LIN {X 0,Y 524.001,Z 252.027,A -85,B 0,C 180,E1 -4869.26,E2 -4869.26} C_VEL
LIN {X 0,Y 524.005,Z 252.027,A -85,B 0,C 180,E1 -4871.738,E2 -4871.738} C_VEL
LIN {X 0,Y 523.995,Z 252.029,A -85,B 0,C 180,E1 -4875.051,E2 -4875.051} C_VEL
LIN {X 0,Y 523.965,Z 252.033,A -85,B 0,C 180,E1 -4877.967,E2 -4877.967} C_VEL
LIN {X 0,Y 523.972,Z 252.031,A -85,B 0,C 180,E1 -4880.408,E2 -4880.408} C_VEL
LIN {X 0,Y 523.916,Z 252.038,A -85,B 0,C 180,E1 -4882.891,E2 -4882.891} C_VEL
LIN {X 0,Y 523.951,Z 252.035,A -85,B 0,C 180,E1 -4885.417,E2 -4885.417} C_VEL
LIN {X 0,Y 523.968,Z 252.033,A -85,B 0,C 180,E1 -4887.997,E2 -4887.997} C_VEL
LIN {X 0,Y 523.943,Z 252.034,A -85,B 0,C 180,E1 -4890.853,E2 -4890.853} C_VEL
LIN {X 0,Y 523.958,Z 252.033,A -85,B 0,C 180,E1 -4893.733,E2 -4893.733} C_VEL
LIN {X 0,Y 523.917,Z 252.038,A -85,B 0,C 180,E1 -4896.402,E2 -4896.402} C_VEL
LIN {X 0,Y 523.925,Z 252.037,A -85,B 0,C 180,E1 -4899.082,E2 -4899.082} C_VEL
LIN {X 0,Y 523.965,Z 252.034,A -85,B 0,C 180,E1 -4901.31,E2 -4901.31} C_VEL
LIN {X 0,Y 523.947,Z 252.035,A -85,B 0,C 180,E1 -4904.689,E2 -4904.689} C_VEL
LIN {X 0,Y 523.916,Z 252.038,A -85,B 0,C 180,E1 -4906.898,E2 -4906.898} C_VEL
LIN {X 0,Y 523.251,Z 252.122,A -85,B 0,C 180,E1 -4907.539,E2 -4907.539} C_VEL
LIN {X 0,Y 520.416,Z 252.476,A -85,B 0,C 180,E1 -4908.581,E2 -4908.581} C_VEL
LIN {X 0,Y 518.018,Z 252.775,A -85,B 0,C 180,E1 -4909.42,E2 -4909.42} C_VEL
LIN {X 0,Y 516.986,Z 252.902,A -85,B 0,C 180,E1 -4910.068,E2 -4910.068} C_VEL
LIN {X 0,Y 516.9,Z 252.911,A -85,B 0,C 180,E1 -4910.287,E2 -4910.287} C_VEL
LIN {X 0,Y 516.875,Z 252.916,A -85,B 0,C 180,E1 -4913.339,E2 -4913.339} C_VEL
LIN {X 0,Y 516.901,Z 252.911,A -85,B 0,C 180,E1 -4916.119,E2 -4916.119} C_VEL
LIN {X 0,Y 516.881,Z 252.915,A -85,B 0,C 180,E1 -4918.933,E2 -4918.933} C_VEL
LIN {X 0,Y 516.911,Z 252.911,A -85,B 0,C 180,E1 -4921.583,E2 -4921.583} C_VEL
LIN {X 0,Y 516.918,Z 252.91,A -85,B 0,C 180,E1 -4924.209,E2 -4924.209} C_VEL
LIN {X 0,Y 516.88,Z 252.916,A -85,B 0,C 180,E1 -4926.776,E2 -4926.776} C_VEL
LIN {X 0,Y 516.923,Z 252.91,A -85,B 0,C 180,E1 -4929.73,E2 -4929.73} C_VEL
LIN {X 0,Y 516.734,Z 252.935,A -85,B 0,C 180,E1 -4932.588,E2 -4932.588} C_VEL
LIN {X 0,Y 516.57,Z 252.955,A -85,B 0,C 180,E1 -4933.398,E2 -4933.398} C_VEL
LIN {X 0,Y 516.586,Z 256.109,A -85,B 0,C 180,E1 -4935.824,E2 -4935.824} C_VEL
LIN {X 0,Y 516.629,Z 259.54,A -85,B 0,C 180,E1 -4938.354,E2 -4938.354} C_VEL
LIN {X 0,Y 516.52,Z 263.691,A -85,B 0,C 180,E1 -4941.391,E2 -4941.391} C_VEL
LIN {X 0,Y 516.557,Z 266.915,A -85,B 0,C 180,E1 -4943.75,E2 -4943.75} C_VEL
LIN {X 0,Y 516.536,Z 270.185,A -85,B 0,C 180,E1 -4946.098,E2 -4946.098} C_VEL
LIN {X 0,Y 516.329,Z 274.545,A -85,B 0,C 180,E1 -4949.219,E2 -4949.219} C_VEL
LIN {X 0,Y 516.246,Z 279.024,A -85,B 0,C 180,E1 -4952.34,E2 -4952.34} C_VEL
LIN {X 0,Y 516.345,Z 280.192,A -85,B 0,C 180,E1 -4953.144,E2 -4953.144} C_VEL
LIN {X 0,Y 517.624,Z 289.128,A -85,B 0,C 180,E1 -4953.453,E2 -4953.453} C_VEL
LIN {X 0,Y 517.444,Z 299.239,A -85,B 0,C 180,E1 -4953.893,E2 -4953.893} C_VEL
LIN {X 0,Y 517.24,Z 307.848,A -85,B 0,C 180,E1 -4954.382,E2 -4954.382} C_VEL
LIN {X 0,Y 517.051,Z 316.077,A -85,B 0,C 180,E1 -4954.97,E2 -4954.97} C_VEL
LIN {X 0,Y 516.884,Z 323.872,A -85,B 0,C 180,E1 -4955.656,E2 -4955.656} C_VEL
LIN {X 0,Y 516.785,Z 331.136,A -85,B 0,C 180,E1 -4956.439,E2 -4956.439} C_VEL
LIN {X 0,Y 516.64,Z 338.552,A -85,B 0,C 180,E1 -4957.424,E2 -4957.424} C_VEL
LIN {X 0,Y 516.488,Z 344.371,A -85,B 0,C 180,E1 -4958.41,E2 -4958.41} C_VEL
LIN {X 0,Y 516.371,Z 348.963,A -85,B 0,C 180,E1 -4959.399,E2 -4959.399} C_VEL
LIN {X 0,Y 516.352,Z 351.937,A -85,B 0,C 180,E1 -4960.191,E2 -4960.191} C_VEL
LIN {X 0,Y 516.316,Z 354.262,A -85,B 0,C 180,E1 -4960.985,E2 -4960.985} C_VEL
LIN {X 0,Y 516.276,Z 355.976,A -85,B 0,C 180,E1 -4961.781,E2 -4961.781} C_VEL
LIN {X 0,Y 516.227,Z 357.177,A -85,B 0,C 180,E1 -4962.58,E2 -4962.58} C_VEL
LIN {X 0,Y 516.198,Z 357.883,A -85,B 0,C 180,E1 -4963.382,E2 -4963.382} C_VEL
LIN {X 0,Y 516.219,Z 358.098,A -85,B 0,C 180,E1 -4964.184,E2 -4964.184} C_VEL
LIN {X 0,Y 516.216,Z 357.765,A -85,B 0,C 180,E1 -4964.99,E2 -4964.99} C_VEL
LIN {X 0,Y 516.236,Z 356.832,A -85,B 0,C 180,E1 -4965.799,E2 -4965.799} C_VEL
LIN {X 0,Y 516.287,Z 354.51,A -85,B 0,C 180,E1 -4967.017,E2 -4967.017} C_VEL
LIN {X 0,Y 516.374,Z 350.713,A -85,B 0,C 180,E1 -4968.241,E2 -4968.241} C_VEL
LIN {X 0,Y 516.445,Z 347.395,A -85,B 0,C 180,E1 -4969.061,E2 -4969.061} C_VEL
LIN {X 0,Y 516.519,Z 343.292,A -85,B 0,C 180,E1 -4969.885,E2 -4969.885} C_VEL
LIN {X 0,Y 516.65,Z 336.774,A -85,B 0,C 180,E1 -4970.92,E2 -4970.92} C_VEL
LIN {X 0,Y 516.798,Z 330.309,A -85,B 0,C 180,E1 -4971.75,E2 -4971.75} C_VEL
LIN {X 0,Y 516.93,Z 324.106,A -85,B 0,C 180,E1 -4972.413,E2 -4972.413} C_VEL
LIN {X 0,Y 517.124,Z 316.421,A -85,B 0,C 180,E1 -4973.094,E2 -4973.094} C_VEL
LIN {X 0,Y 517.321,Z 309.115,A -85,B 0,C 180,E1 -4973.625,E2 -4973.625} C_VEL
LIN {X 0,Y 517.474,Z 300.931,A -85,B 0,C 180,E1 -4974.109,E2 -4974.109} C_VEL
LIN {X 0,Y 517.594,Z 291.635,A -85,B 0,C 180,E1 -4974.537,E2 -4974.537} C_VEL
LIN {X 0,Y 517.263,Z 285.961,A -85,B 0,C 180,E1 -4974.75,E2 -4974.75} C_VEL
LIN {X 0,Y 516.275,Z 280.189,A -85,B 0,C 180,E1 -4974.96,E2 -4974.96} C_VEL
LIN {X 0,Y 516.296,Z 275.269,A -85,B 0,C 180,E1 -4978.451,E2 -4978.451} C_VEL
LIN {X 0,Y 516.338,Z 271.494,A -85,B 0,C 180,E1 -4981.145,E2 -4981.145} C_VEL
LIN {X 0,Y 516.359,Z 267.678,A -85,B 0,C 180,E1 -4983.919,E2 -4983.919} C_VEL
LIN {X 0,Y 516.405,Z 263.771,A -85,B 0,C 180,E1 -4986.784,E2 -4986.784} C_VEL
LIN {X 0,Y 516.448,Z 259.768,A -85,B 0,C 180,E1 -4989.76,E2 -4989.76} C_VEL
LIN {X 0,Y 516.585,Z 255.637,A -85,B 0,C 180,E1 -4992.86,E2 -4992.86} C_VEL
LIN {X 0,Y 516.633,Z 252.947,A -85,B 0,C 180,E1 -4995.02,E2 -4995.02} C_VEL
LIN {X 0,Y 516.837,Z 252.916,A -85,B 0,C 180,E1 -4997.246,E2 -4997.246} C_VEL
LIN {X 0,Y 516.887,Z 252.916,A -85,B 0,C 180,E1 -4999.587,E2 -4999.587} C_VEL
LIN {X 0,Y 516.85,Z 252.917,A -85,B 0,C 180,E1 -5002.276,E2 -5002.276} C_VEL
LIN {X 0,Y 516.876,Z 252.912,A -85,B 0,C 180,E1 -5005.177,E2 -5005.177} C_VEL
LIN {X 0,Y 516.856,Z 252.915,A -85,B 0,C 180,E1 -5007.976,E2 -5007.976} C_VEL
LIN {X 0,Y 516.904,Z 252.912,A -85,B 0,C 180,E1 -5010.697,E2 -5010.697} C_VEL
LIN {X 0,Y 516.925,Z 252.91,A -85,B 0,C 180,E1 -5013.805,E2 -5013.805} C_VEL
LIN {X 0,Y 516.847,Z 252.918,A -85,B 0,C 180,E1 -5016.777,E2 -5016.777} C_VEL
LIN {X 0,Y 516.923,Z 252.906,A -85,B 0,C 180,E1 -5019.733,E2 -5019.733} C_VEL
LIN {X 0,Y 516.915,Z 252.905,A -85,B 0,C 180,E1 -5022.598,E2 -5022.598} C_VEL
LIN {X 0,Y 516.925,Z 252.908,A -85,B 0,C 180,E1 -5025.031,E2 -5025.031} C_VEL
LIN {X 0,Y 516.99,Z 252.9,A -85,B 0,C 180,E1 -5028.236,E2 -5028.236} C_VEL
LIN {X 0,Y 516.953,Z 252.905,A -85,B 0,C 180,E1 -5031.401,E2 -5031.401} C_VEL
LIN {X 0,Y 517.009,Z 252.898,A -85,B 0,C 180,E1 -5034.541,E2 -5034.541} C_VEL
LIN {X 0,Y 517.074,Z 252.89,A -85,B 0,C 180,E1 -5037.665,E2 -5037.665} C_VEL
LIN {X 0,Y 517.082,Z 252.89,A -85,B 0,C 180,E1 -5040.78,E2 -5040.78} C_VEL
LIN {X 0,Y 517.001,Z 252.896,A -85,B 0,C 180,E1 -5043.118,E2 -5043.118} C_VEL
LIN {X 0,Y 517.002,Z 252.894,A -85,B 0,C 180,E1 -5046.245,E2 -5046.245} C_VEL
LIN {X 0,Y 516.933,Z 252.904,A -85,B 0,C 180,E1 -5049.391,E2 -5049.391} C_VEL
LIN {X 0,Y 516.974,Z 252.905,A -85,B 0,C 180,E1 -5051.825,E2 -5051.825} C_VEL
LIN {X 0,Y 516.935,Z 252.908,A -85,B 0,C 180,E1 -5055.148,E2 -5055.148} C_VEL
LIN {X 0,Y 516.903,Z 252.913,A -85,B 0,C 180,E1 -5058.224,E2 -5058.224} C_VEL
LIN {X 0,Y 516.903,Z 252.909,A -85,B 0,C 180,E1 -5060.703,E2 -5060.703} C_VEL
LIN {X 0,Y 516.904,Z 252.91,A -85,B 0,C 180,E1 -5064.073,E2 -5064.073} C_VEL
LIN {X 0,Y 516.889,Z 252.911,A -85,B 0,C 180,E1 -5066.661,E2 -5066.661} C_VEL
LIN {X 0,Y 516.903,Z 252.912,A -85,B 0,C 180,E1 -5069.525,E2 -5069.525} C_VEL
LIN {X 0,Y 516.894,Z 252.915,A -85,B 0,C 180,E1 -5072.546,E2 -5072.546} C_VEL
LIN {X 0,Y 516.857,Z 252.919,A -85,B 0,C 180,E1 -5075.331,E2 -5075.331} C_VEL
LIN {X 0,Y 516.88,Z 252.917,A -85,B 0,C 180,E1 -5078.717,E2 -5078.717} C_VEL
LIN {X 0,Y 516.911,Z 252.912,A -85,B 0,C 180,E1 -5081.776,E2 -5081.776} C_VEL
LIN {X 0,Y 516.89,Z 252.918,A -85,B 0,C 180,E1 -5085.008,E2 -5085.008} C_VEL
LIN {X 0,Y 516.913,Z 252.912,A -85,B 0,C 180,E1 -5088.4,E2 -5088.4} C_VEL
LIN {X 0,Y 516.875,Z 252.917,A -85,B 0,C 180,E1 -5091.285,E2 -5091.285} C_VEL
LIN {X 0,Y 516.869,Z 252.918,A -85,B 0,C 180,E1 -5094.221,E2 -5094.221} C_VEL
LIN {X 0,Y 516.898,Z 252.925,A -85,B 0,C 180,E1 -5094.898,E2 -5094.898} C_VEL
LIN {X 0,Y 517.688,Z 257.17,A -85,B 0,C 180,E1 -5096.647,E2 -5096.647} C_VEL
LIN {X 0,Y 517.651,Z 262.78,A -85,B 0,C 180,E1 -5098.797,E2 -5098.797} C_VEL
LIN {X 0,Y 517.346,Z 271.703,A -85,B 0,C 180,E1 -5102.008,E2 -5102.008} C_VEL
LIN {X 0,Y 517.053,Z 280.514,A -85,B 0,C 180,E1 -5105.081,E2 -5105.081} C_VEL
LIN {X 0,Y 516.846,Z 289.348,A -85,B 0,C 180,E1 -5108.042,E2 -5108.042} C_VEL
LIN {X 0,Y 516.671,Z 299.586,A -85,B 0,C 180,E1 -5111.359,E2 -5111.359} C_VEL
LIN {X 0,Y 516.561,Z 309.871,A -85,B 0,C 180,E1 -5114.616,E2 -5114.616} C_VEL
LIN {X 0,Y 516.453,Z 320.168,A -85,B 0,C 180,E1 -5117.824,E2 -5117.824} C_VEL
LIN {X 0,Y 516.452,Z 324.035,A -85,B 0,C 180,E1 -5119.018,E2 -5119.018} C_VEL
LIN {X 0,Y 517.543,Z 335.925,A -85,B 0,C 180,E1 -5119.388,E2 -5119.388} C_VEL
LIN {X 0,Y 517.369,Z 346.244,A -85,B 0,C 180,E1 -5119.83,E2 -5119.83} C_VEL
LIN {X 0,Y 517.182,Z 354.979,A -85,B 0,C 180,E1 -5120.32,E2 -5120.32} C_VEL
LIN {X 0,Y 516.995,Z 363.323,A -85,B 0,C 180,E1 -5120.909,E2 -5120.909} C_VEL
LIN {X 0,Y 516.826,Z 371.224,A -85,B 0,C 180,E1 -5121.595,E2 -5121.595} C_VEL
LIN {X 0,Y 516.652,Z 378.613,A -85,B 0,C 180,E1 -5122.38,E2 -5122.38} C_VEL
LIN {X 0,Y 516.528,Z 385.999,A -85,B 0,C 180,E1 -5123.343,E2 -5123.343} C_VEL
LIN {X 0,Y 516.449,Z 392.004,A -85,B 0,C 180,E1 -5124.339,E2 -5124.339} C_VEL
LIN {X 0,Y 516.312,Z 396.638,A -85,B 0,C 180,E1 -5125.316,E2 -5125.316} C_VEL
LIN {X 0,Y 516.361,Z 399.657,A -85,B 0,C 180,E1 -5126.099,E2 -5126.099} C_VEL
LIN {X 0,Y 516.294,Z 401.992,A -85,B 0,C 180,E1 -5126.88,E2 -5126.88} C_VEL
LIN {X 0,Y 516.263,Z 403.75,A -85,B 0,C 180,E1 -5127.66,E2 -5127.66} C_VEL
LIN {X 0,Y 516.191,Z 405.007,A -85,B 0,C 180,E1 -5128.441,E2 -5128.441} C_VEL
LIN {X 0,Y 516.16,Z 405.791,A -85,B 0,C 180,E1 -5129.221,E2 -5129.221} C_VEL
LIN {X 0,Y 516.16,Z 406.089,A -85,B 0,C 180,E1 -5130.001,E2 -5130.001} C_VEL
LIN {X 0,Y 516.16,Z 405.792,A -85,B 0,C 180,E1 -5130.781,E2 -5130.781} C_VEL
LIN {X 0,Y 516.191,Z 405.009,A -85,B 0,C 180,E1 -5131.561,E2 -5131.561} C_VEL
LIN {X 0,Y 516.263,Z 403.752,A -85,B 0,C 180,E1 -5132.342,E2 -5132.342} C_VEL
LIN {X 0,Y 516.323,Z 400.836,A -85,B 0,C 180,E1 -5133.513,E2 -5133.513} C_VEL
LIN {X 0,Y 516.342,Z 398.176,A -85,B 0,C 180,E1 -5134.294,E2 -5134.294} C_VEL
LIN {X 0,Y 516.425,Z 392.973,A -85,B 0,C 180,E1 -5135.467,E2 -5135.467} C_VEL
LIN {X 0,Y 516.507,Z 387.575,A -85,B 0,C 180,E1 -5136.414,E2 -5136.414} C_VEL
LIN {X 0,Y 516.626,Z 380.33,A -85,B 0,C 180,E1 -5137.426,E2 -5137.426} C_VEL
LIN {X 0,Y 516.829,Z 372.266,A -85,B 0,C 180,E1 -5138.308,E2 -5138.308} C_VEL
LIN {X 0,Y 516.958,Z 364.569,A -85,B 0,C 180,E1 -5138.996,E2 -5138.996} C_VEL
LIN {X 0,Y 517.141,Z 356.49,A -85,B 0,C 180,E1 -5139.584,E2 -5139.584} C_VEL
LIN {X 0,Y 517.375,Z 348.126,A -85,B 0,C 180,E1 -5140.073,E2 -5140.073} C_VEL
LIN {X 0,Y 517.486,Z 339.588,A -85,B 0,C 180,E1 -5140.467,E2 -5140.467} C_VEL
LIN {X 0,Y 517.348,Z 332.736,A -85,B 0,C 180,E1 -5140.717,E2 -5140.717} C_VEL
LIN {X 0,Y 516.423,Z 324.083,A -85,B 0,C 180,E1 -5140.984,E2 -5140.984} C_VEL
LIN {X 0,Y 516.495,Z 313.787,A -85,B 0,C 180,E1 -5144.178,E2 -5144.178} C_VEL
LIN {X 0,Y 516.569,Z 304.8,A -85,B 0,C 180,E1 -5147.009,E2 -5147.009} C_VEL
LIN {X 0,Y 516.707,Z 295.849,A -85,B 0,C 180,E1 -5149.88,E2 -5149.88} C_VEL
LIN {X 0,Y 516.931,Z 286.915,A -85,B 0,C 180,E1 -5152.798,E2 -5152.798} C_VEL
LIN {X 0,Y 517.115,Z 278.013,A -85,B 0,C 180,E1 -5155.78,E2 -5155.78} C_VEL
LIN {X 0,Y 517.404,Z 269.157,A -85,B 0,C 180,E1 -5158.83,E2 -5158.83} C_VEL
LIN {X 0,Y 517.663,Z 260.359,A -85,B 0,C 180,E1 -5161.971,E2 -5161.971} C_VEL
LIN {X 0,Y 517.557,Z 256.603,A -85,B 0,C 180,E1 -5163.365,E2 -5163.365} C_VEL
LIN {X 0,Y 516.905,Z 252.913,A -85,B 0,C 180,E1 -5164.824,E2 -5164.824} C_VEL
LIN {X 0,Y 516.887,Z 252.914,A -85,B 0,C 180,E1 -5167.943,E2 -5167.943} C_VEL
LIN {X 0,Y 516.89,Z 252.913,A -85,B 0,C 180,E1 -5170.742,E2 -5170.742} C_VEL
LIN {X 0,Y 516.89,Z 252.912,A -85,B 0,C 180,E1 -5172.832,E2 -5172.832} C_VEL
LIN {X 0,Y 516.903,Z 252.91,A -85,B 0,C 180,E1 -5175.007,E2 -5175.007} C_VEL
LIN {X 0,Y 516.921,Z 252.911,A -85,B 0,C 180,E1 -5178.399,E2 -5178.399} C_VEL
LIN {X 0,Y 516.887,Z 252.914,A -85,B 0,C 180,E1 -5181.284,E2 -5181.284} C_VEL
LIN {X 0,Y 516.876,Z 252.916,A -85,B 0,C 180,E1 -5184.219,E2 -5184.219} C_VEL
LIN {X 0,Y 516.903,Z 252.911,A -85,B 0,C 180,E1 -5187.053,E2 -5187.053} C_VEL
LIN {X 0,Y 516.9,Z 252.913,A -85,B 0,C 180,E1 -5189.796,E2 -5189.796} C_VEL
LIN {X 0,Y 516.933,Z 252.908,A -85,B 0,C 180,E1 -5192.467,E2 -5192.467} C_VEL
LIN {X 0,Y 516.884,Z 252.914,A -85,B 0,C 180,E1 -5195.07,E2 -5195.07} C_VEL
LIN {X 0,Y 516.877,Z 252.917,A -85,B 0,C 180,E1 -5197.621,E2 -5197.621} C_VEL
LIN {X 0,Y 516.94,Z 252.906,A -85,B 0,C 180,E1 -5200.129,E2 -5200.129} C_VEL
LIN {X 0,Y 516.913,Z 252.91,A -85,B 0,C 180,E1 -5202.595,E2 -5202.595} C_VEL
LIN {X 0,Y 516.949,Z 252.907,A -85,B 0,C 180,E1 -5205.029,E2 -5205.029} C_VEL
LIN {X 0,Y 516.974,Z 252.902,A -85,B 0,C 180,E1 -5208.233,E2 -5208.233} C_VEL
LIN {X 0,Y 516.962,Z 252.904,A -85,B 0,C 180,E1 -5211.398,E2 -5211.398} C_VEL
LIN {X 0,Y 517.007,Z 252.899,A -85,B 0,C 180,E1 -5213.756,E2 -5213.756} C_VEL
LIN {X 0,Y 517.018,Z 252.899,A -85,B 0,C 180,E1 -5216.882,E2 -5216.882} C_VEL
LIN {X 0,Y 517.09,Z 252.889,A -85,B 0,C 180,E1 -5219.999,E2 -5219.999} C_VEL
LIN {X 0,Y 517.018,Z 252.897,A -85,B 0,C 180,E1 -5223.115,E2 -5223.115} C_VEL
LIN {X 0,Y 517.015,Z 252.899,A -85,B 0,C 180,E1 -5226.242,E2 -5226.242} C_VEL
LIN {X 0,Y 516.955,Z 252.905,A -85,B 0,C 180,E1 -5229.388,E2 -5229.388} C_VEL
LIN {X 0,Y 516.955,Z 252.905,A -85,B 0,C 180,E1 -5231.805,E2 -5231.805} C_VEL
LIN {X 0,Y 516.946,Z 252.907,A -85,B 0,C 180,E1 -5235.145,E2 -5235.145} C_VEL
LIN {X 0,Y 516.926,Z 252.91,A -85,B 0,C 180,E1 -5238.22,E2 -5238.22} C_VEL
LIN {X 0,Y 516.912,Z 252.91,A -85,B 0,C 180,E1 -5240.7,E2 -5240.7} C_VEL
LIN {X 0,Y 516.91,Z 252.912,A -85,B 0,C 180,E1 -5244.07,E2 -5244.07} C_VEL
LIN {X 0,Y 516.925,Z 252.908,A -85,B 0,C 180,E1 -5246.656,E2 -5246.656} C_VEL
LIN {X 0,Y 516.908,Z 252.912,A -85,B 0,C 180,E1 -5249.522,E2 -5249.522} C_VEL
LIN {X 0,Y 516.897,Z 252.912,A -85,B 0,C 180,E1 -5252.542,E2 -5252.542} C_VEL
LIN {X 0,Y 516.878,Z 252.917,A -85,B 0,C 180,E1 -5255.33,E2 -5255.33} C_VEL
LIN {X 0,Y 516.875,Z 252.915,A -85,B 0,C 180,E1 -5257.941,E2 -5257.941} C_VEL
LIN {X 0,Y 516.897,Z 252.913,A -85,B 0,C 180,E1 -5260.738,E2 -5260.738} C_VEL
LIN {X 0,Y 516.874,Z 252.915,A -85,B 0,C 180,E1 -5263.901,E2 -5263.901} C_VEL
LIN {X 0,Y 516.874,Z 252.915,A -85,B 0,C 180,E1 -5266.105,E2 -5266.105} C_VEL
LIN {X 0,Y 516.898,Z 252.913,A -85,B 0,C 180,E1 -5269.259,E2 -5269.259} C_VEL
LIN {X 0,Y 516.9,Z 252.911,A -85,B 0,C 180,E1 -5270.287,E2 -5270.287} C_VEL
LIN {X 0,Y 516.23,Z 252.996,A -85,B 0,C 180,E1 -5270.937,E2 -5270.937} C_VEL
LIN {X 0,Y 513.374,Z 253.353,A -85,B 0,C 180,E1 -5271.992,E2 -5271.992} C_VEL
LIN {X 0,Y 510.957,Z 253.655,A -85,B 0,C 180,E1 -5272.842,E2 -5272.842} C_VEL
LIN {X 0,Y 509.911,Z 253.784,A -85,B 0,C 180,E1 -5273.498,E2 -5273.498} C_VEL
LIN {X 0,Y 509.822,Z 253.793,A -85,B 0,C 180,E1 -5273.721,E2 -5273.721} C_VEL
LIN {X 0,Y 509.851,Z 253.791,A -85,B 0,C 180,E1 -5276.538,E2 -5276.538} C_VEL
LIN {X 0,Y 509.837,Z 253.793,A -85,B 0,C 180,E1 -5279.333,E2 -5279.333} C_VEL
LIN {X 0,Y 509.881,Z 253.786,A -85,B 0,C 180,E1 -5282.053,E2 -5282.053} C_VEL
LIN {X 0,Y 509.865,Z 253.79,A -85,B 0,C 180,E1 -5284.702,E2 -5284.702} C_VEL
LIN {X 0,Y 509.867,Z 253.788,A -85,B 0,C 180,E1 -5287.441,E2 -5287.441} C_VEL
LIN {X 0,Y 509.899,Z 253.785,A -85,B 0,C 180,E1 -5289.843,E2 -5289.843} C_VEL
LIN {X 0,Y 509.731,Z 253.807,A -85,B 0,C 180,E1 -5292.341,E2 -5292.341} C_VEL
LIN {X 0,Y 509.561,Z 253.827,A -85,B 0,C 180,E1 -5293.163,E2 -5293.163} C_VEL
LIN {X 0,Y 509.492,Z 254.335,A -85,B 0,C 180,E1 -5293.984,E2 -5293.984} C_VEL
LIN {X 0,Y 509.493,Z 257.625,A -85,B 0,C 180,E1 -5296.437,E2 -5296.437} C_VEL
LIN {X 0,Y 509.501,Z 260.888,A -85,B 0,C 180,E1 -5298.864,E2 -5298.864} C_VEL
LIN {X 0,Y 509.425,Z 265.235,A -85,B 0,C 180,E1 -5302.069,E2 -5302.069} C_VEL
LIN {X 0,Y 509.508,Z 267.408,A -85,B 0,C 180,E1 -5303.664,E2 -5303.664} C_VEL
LIN {X 0,Y 509.453,Z 270.692,A -85,B 0,C 180,E1 -5306.044,E2 -5306.044} C_VEL
LIN {X 0,Y 509.252,Z 275.102,A -85,B 0,C 180,E1 -5309.208,E2 -5309.208} C_VEL
LIN {X 0,Y 509.258,Z 280.437,A -85,B 0,C 180,E1 -5312.965,E2 -5312.965} C_VEL
LIN {X 0,Y 510.305,Z 286.696,A -85,B 0,C 180,E1 -5313.206,E2 -5313.206} C_VEL
LIN {X 0,Y 510.627,Z 291.745,A -85,B 0,C 180,E1 -5313.402,E2 -5313.402} C_VEL
LIN {X 0,Y 510.464,Z 299.482,A -85,B 0,C 180,E1 -5313.749,E2 -5313.749} C_VEL
LIN {X 0,Y 510.261,Z 308.102,A -85,B 0,C 180,E1 -5314.245,E2 -5314.245} C_VEL
LIN {X 0,Y 510.059,Z 316.344,A -85,B 0,C 180,E1 -5314.84,E2 -5314.84} C_VEL
LIN {X 0,Y 509.868,Z 324.153,A -85,B 0,C 180,E1 -5315.536,E2 -5315.536} C_VEL
LIN {X 0,Y 509.746,Z 331.438,A -85,B 0,C 180,E1 -5316.331,E2 -5316.331} C_VEL
LIN {X 0,Y 509.606,Z 338.846,A -85,B 0,C 180,E1 -5317.328,E2 -5317.328} C_VEL
LIN {X 0,Y 509.443,Z 344.674,A -85,B 0,C 180,E1 -5318.328,E2 -5318.328} C_VEL
LIN {X 0,Y 509.337,Z 348.485,A -85,B 0,C 180,E1 -5319.129,E2 -5319.129} C_VEL
LIN {X 0,Y 509.272,Z 352.834,A -85,B 0,C 180,E1 -5320.334,E2 -5320.334} C_VEL
LIN {X 0,Y 509.233,Z 355.846,A -85,B 0,C 180,E1 -5321.526,E2 -5321.526} C_VEL
LIN {X 0,Y 509.192,Z 356.701,A -85,B 0,C 180,E1 -5321.947,E2 -5321.947} C_VEL
LIN {X 0,Y 509.136,Z 357.747,A -85,B 0,C 180,E1 -5322.758,E2 -5322.758} C_VEL
LIN {X 0,Y 509.104,Z 358.292,A -85,B 0,C 180,E1 -5323.572,E2 -5323.572} C_VEL
LIN {X 0,Y 509.147,Z 358.126,A -85,B 0,C 180,E1 -5324.94,E2 -5324.94} C_VEL
LIN {X 0,Y 509.164,Z 356.91,A -85,B 0,C 180,E1 -5326.024,E2 -5326.024} C_VEL
LIN {X 0,Y 509.238,Z 354.286,A -85,B 0,C 180,E1 -5327.26,E2 -5327.26} C_VEL
LIN {X 0,Y 509.294,Z 351.801,A -85,B 0,C 180,E1 -5328.099,E2 -5328.099} C_VEL
LIN {X 0,Y 509.366,Z 348.684,A -85,B 0,C 180,E1 -5328.918,E2 -5328.918} C_VEL
LIN {X 0,Y 509.458,Z 343.647,A -85,B 0,C 180,E1 -5329.963,E2 -5329.963} C_VEL
LIN {X 0,Y 509.626,Z 337.138,A -85,B 0,C 180,E1 -5331.01,E2 -5331.01} C_VEL
LIN {X 0,Y 509.77,Z 330.676,A -85,B 0,C 180,E1 -5331.852,E2 -5331.852} C_VEL
LIN {X 0,Y 509.923,Z 323.971,A -85,B 0,C 180,E1 -5332.575,E2 -5332.575} C_VEL
LIN {X 0,Y 510.117,Z 316.671,A -85,B 0,C 180,E1 -5333.226,E2 -5333.226} C_VEL
LIN {X 0,Y 510.324,Z 309.507,A -85,B 0,C 180,E1 -5333.753,E2 -5333.753} C_VEL
LIN {X 0,Y 510.511,Z 300.587,A -85,B 0,C 180,E1 -5334.284,E2 -5334.284} C_VEL
LIN {X 0,Y 510.662,Z 290.756,A -85,B 0,C 180,E1 -5334.731,E2 -5334.731} C_VEL
LIN {X 0,Y 509.759,Z 283.857,A -85,B 0,C 180,E1 -5334.984,E2 -5334.984} C_VEL
LIN {X 0,Y 509.205,Z 280.518,A -85,B 0,C 180,E1 -5335.117,E2 -5335.117} C_VEL
LIN {X 0,Y 509.215,Z 276.475,A -85,B 0,C 180,E1 -5337.985,E2 -5337.985} C_VEL
LIN {X 0,Y 509.262,Z 272.044,A -85,B 0,C 180,E1 -5341.176,E2 -5341.176} C_VEL
LIN {X 0,Y 509.296,Z 268.029,A -85,B 0,C 180,E1 -5344.114,E2 -5344.114} C_VEL
LIN {X 0,Y 509.363,Z 264.365,A -85,B 0,C 180,E1 -5346.849,E2 -5346.849} C_VEL
LIN {X 0,Y 509.382,Z 260.939,A -85,B 0,C 180,E1 -5349.412,E2 -5349.412} C_VEL
LIN {X 0,Y 509.501,Z 256.841,A -85,B 0,C 180,E1 -5352.522,E2 -5352.522} C_VEL
LIN {X 0,Y 509.568,Z 254.029,A -85,B 0,C 180,E1 -5354.698,E2 -5354.698} C_VEL
LIN {X 0,Y 509.794,Z 253.794,A -85,B 0,C 180,E1 -5357.509,E2 -5357.509} C_VEL
LIN {X 0,Y 509.845,Z 253.788,A -85,B 0,C 180,E1 -5360.526,E2 -5360.526} C_VEL
LIN {X 0,Y 509.817,Z 253.792,A -85,B 0,C 180,E1 -5363.649,E2 -5363.649} C_VEL
LIN {X 0,Y 509.842,Z 253.788,A -85,B 0,C 180,E1 -5366.54,E2 -5366.54} C_VEL
LIN {X 0,Y 509.826,Z 253.792,A -85,B 0,C 180,E1 -5369.335,E2 -5369.335} C_VEL
LIN {X 0,Y 509.876,Z 253.787,A -85,B 0,C 180,E1 -5372.056,E2 -5372.056} C_VEL
LIN {X 0,Y 509.858,Z 253.786,A -85,B 0,C 180,E1 -5374.705,E2 -5374.705} C_VEL
LIN {X 0,Y 509.809,Z 253.793,A -85,B 0,C 180,E1 -5377.459,E2 -5377.459} C_VEL
LIN {X 0,Y 509.901,Z 253.782,A -85,B 0,C 180,E1 -5379.846,E2 -5379.846} C_VEL
LIN {X 0,Y 509.87,Z 253.787,A -85,B 0,C 180,E1 -5383.176,E2 -5383.176} C_VEL
LIN {X 0,Y 509.846,Z 253.786,A -85,B 0,C 180,E1 -5385.635,E2 -5385.635} C_VEL
LIN {X 0,Y 509.912,Z 253.778,A -85,B 0,C 180,E1 -5388.876,E2 -5388.876} C_VEL
LIN {X 0,Y 509.936,Z 253.776,A -85,B 0,C 180,E1 -5392.08,E2 -5392.08} C_VEL
LIN {X 0,Y 509.96,Z 253.778,A -85,B 0,C 180,E1 -5394.466,E2 -5394.466} C_VEL
LIN {X 0,Y 510.045,Z 253.765,A -85,B 0,C 180,E1 -5397.632,E2 -5397.632} C_VEL
LIN {X 0,Y 510.052,Z 253.765,A -85,B 0,C 180,E1 -5400.791,E2 -5400.791} C_VEL
LIN {X 0,Y 509.943,Z 253.775,A -85,B 0,C 180,E1 -5403.162,E2 -5403.162} C_VEL
LIN {X 0,Y 509.97,Z 253.77,A -85,B 0,C 180,E1 -5406.331,E2 -5406.331} C_VEL
LIN {X 0,Y 509.901,Z 253.785,A -85,B 0,C 180,E1 -5408.722,E2 -5408.722} C_VEL
LIN {X 0,Y 509.942,Z 253.78,A -85,B 0,C 180,E1 -5411.932,E2 -5411.932} C_VEL
LIN {X 0,Y 509.885,Z 253.785,A -85,B 0,C 180,E1 -5415.243,E2 -5415.243} C_VEL
LIN {X 0,Y 509.852,Z 253.791,A -85,B 0,C 180,E1 -5417.993,E2 -5417.993} C_VEL
LIN {X 0,Y 509.878,Z 253.783,A -85,B 0,C 180,E1 -5420.403,E2 -5420.403} C_VEL
LIN {X 0,Y 509.829,Z 253.79,A -85,B 0,C 180,E1 -5423.565,E2 -5423.565} C_VEL
LIN {X 0,Y 509.876,Z 253.787,A -85,B 0,C 180,E1 -5426.374,E2 -5426.374} C_VEL
LIN {X 0,Y 509.85,Z 253.789,A -85,B 0,C 180,E1 -5429.752,E2 -5429.752} C_VEL
LIN {X 0,Y 509.87,Z 253.788,A -85,B 0,C 180,E1 -5432.776,E2 -5432.776} C_VEL
LIN {X 0,Y 509.816,Z 253.798,A -85,B 0,C 180,E1 -5435.579,E2 -5435.579} C_VEL
LIN {X 0,Y 509.846,Z 253.79,A -85,B 0,C 180,E1 -5438.339,E2 -5438.339} C_VEL
LIN {X 0,Y 509.858,Z 253.787,A -85,B 0,C 180,E1 -5441.426,E2 -5441.426} C_VEL
LIN {X 0,Y 509.834,Z 253.793,A -85,B 0,C 180,E1 -5444.671,E2 -5444.671} C_VEL
LIN {X 0,Y 509.855,Z 253.793,A -85,B 0,C 180,E1 -5448.104,E2 -5448.104} C_VEL
LIN {X 0,Y 509.842,Z 253.79,A -85,B 0,C 180,E1 -5450.649,E2 -5450.649} C_VEL
LIN {X 0,Y 509.821,Z 253.794,A -85,B 0,C 180,E1 -5453.648,E2 -5453.648} C_VEL
LIN {X 0,Y 509.871,Z 253.98,A -85,B 0,C 180,E1 -5454.748,E2 -5454.748} C_VEL
LIN {X 0,Y 510.712,Z 258.417,A -85,B 0,C 180,E1 -5456.604,E2 -5456.604} C_VEL
LIN {X 0,Y 510.706,Z 263.38,A -85,B 0,C 180,E1 -5458.563,E2 -5458.563} C_VEL
LIN {X 0,Y 510.338,Z 272.215,A -85,B 0,C 180,E1 -5461.808,E2 -5461.808} C_VEL
LIN {X 0,Y 510.012,Z 281.573,A -85,B 0,C 180,E1 -5465.123,E2 -5465.123} C_VEL
LIN {X 0,Y 509.774,Z 290.457,A -85,B 0,C 180,E1 -5468.148,E2 -5468.148} C_VEL
LIN {X 0,Y 509.607,Z 299.341,A -85,B 0,C 180,E1 -5471.091,E2 -5471.091} C_VEL
LIN {X 0,Y 509.493,Z 309.604,A -85,B 0,C 180,E1 -5474.397,E2 -5474.397} C_VEL
LIN {X 0,Y 509.342,Z 318.558,A -85,B 0,C 180,E1 -5477.247,E2 -5477.247} C_VEL
LIN {X 0,Y 509.366,Z 323.694,A -85,B 0,C 180,E1 -5478.864,E2 -5478.864} C_VEL
LIN {X 0,Y 510.524,Z 336.827,A -85,B 0,C 180,E1 -5479.291,E2 -5479.291} C_VEL
LIN {X 0,Y 510.361,Z 345.901,A -85,B 0,C 180,E1 -5479.689,E2 -5479.689} C_VEL
LIN {X 0,Y 510.187,Z 354.638,A -85,B 0,C 180,E1 -5480.186,E2 -5480.186} C_VEL
LIN {X 0,Y 509.97,Z 362.983,A -85,B 0,C 180,E1 -5480.782,E2 -5480.782} C_VEL
LIN {X 0,Y 509.799,Z 370.885,A -85,B 0,C 180,E1 -5481.479,E2 -5481.479} C_VEL
LIN {X 0,Y 509.586,Z 378.274,A -85,B 0,C 180,E1 -5482.273,E2 -5482.273} C_VEL
LIN {X 0,Y 509.427,Z 386.444,A -85,B 0,C 180,E1 -5483.368,E2 -5483.368} C_VEL
LIN {X 0,Y 509.342,Z 392.633,A -85,B 0,C 180,E1 -5484.458,E2 -5484.458} C_VEL
LIN {X 0,Y 509.236,Z 397.836,A -85,B 0,C 180,E1 -5485.648,E2 -5485.648} C_VEL
LIN {X 0,Y 509.243,Z 400.499,A -85,B 0,C 180,E1 -5486.44,E2 -5486.44} C_VEL
LIN {X 0,Y 509.192,Z 403.42,A -85,B 0,C 180,E1 -5487.628,E2 -5487.628} C_VEL
LIN {X 0,Y 509.112,Z 404.677,A -85,B 0,C 180,E1 -5488.419,E2 -5488.419} C_VEL
LIN {X 0,Y 509.073,Z 405.461,A -85,B 0,C 180,E1 -5489.21,E2 -5489.21} C_VEL
LIN {X 0,Y 509.071,Z 405.759,A -85,B 0,C 180,E1 -5490.001,E2 -5490.001} C_VEL
LIN {X 0,Y 509.073,Z 405.464,A -85,B 0,C 180,E1 -5490.792,E2 -5490.792} C_VEL
LIN {X 0,Y 509.112,Z 404.681,A -85,B 0,C 180,E1 -5491.583,E2 -5491.583} C_VEL
LIN {X 0,Y 509.192,Z 403.424,A -85,B 0,C 180,E1 -5492.374,E2 -5492.374} C_VEL
LIN {X 0,Y 509.244,Z 400.508,A -85,B 0,C 180,E1 -5493.562,E2 -5493.562} C_VEL
LIN {X 0,Y 509.236,Z 397.846,A -85,B 0,C 180,E1 -5494.354,E2 -5494.354} C_VEL
LIN {X 0,Y 509.342,Z 392.644,A -85,B 0,C 180,E1 -5495.544,E2 -5495.544} C_VEL
LIN {X 0,Y 509.482,Z 386.125,A -85,B 0,C 180,E1 -5496.685,E2 -5496.685} C_VEL
LIN {X 0,Y 509.592,Z 378.294,A -85,B 0,C 180,E1 -5497.729,E2 -5497.729} C_VEL
LIN {X 0,Y 509.801,Z 370.91,A -85,B 0,C 180,E1 -5498.523,E2 -5498.523} C_VEL
LIN {X 0,Y 509.973,Z 363.004,A -85,B 0,C 180,E1 -5499.22,E2 -5499.22} C_VEL
LIN {X 0,Y 510.152,Z 354.654,A -85,B 0,C 180,E1 -5499.817,E2 -5499.817} C_VEL
LIN {X 0,Y 510.424,Z 344,A -85,B 0,C 180,E1 -5500.412,E2 -5500.412} C_VEL
LIN {X 0,Y 510.412,Z 334.072,A -85,B 0,C 180,E1 -5500.814,E2 -5500.814} C_VEL
LIN {X 0,Y 509.327,Z 323.753,A -85,B 0,C 180,E1 -5501.139,E2 -5501.139} C_VEL
LIN {X 0,Y 509.424,Z 314.809,A -85,B 0,C 180,E1 -5503.972,E2 -5503.972} C_VEL
LIN {X 0,Y 509.482,Z 305.849,A -85,B 0,C 180,E1 -5506.84,E2 -5506.84} C_VEL
LIN {X 0,Y 509.629,Z 296.914,A -85,B 0,C 180,E1 -5509.748,E2 -5509.748} C_VEL
LIN {X 0,Y 509.869,Z 287.991,A -85,B 0,C 180,E1 -5512.704,E2 -5512.704} C_VEL
LIN {X 0,Y 510.074,Z 279.105,A -85,B 0,C 180,E1 -5515.724,E2 -5515.724} C_VEL
LIN {X 0,Y 510.288,Z 272.045,A -85,B 0,C 180,E1 -5518.182,E2 -5518.182} C_VEL
LIN {X 0,Y 510.591,Z 264.124,A -85,B 0,C 180,E1 -5521.018,E2 -5521.018} C_VEL
LIN {X 0,Y 510.655,Z 259.011,A -85,B 0,C 180,E1 -5522.909,E2 -5522.909} C_VEL
LIN {X 0,Y 509.864,Z 253.79,A -85,B 0,C 180,E1 -5525.014,E2 -5525.014} C_VEL
LIN {X 0,Y 509.857,Z 253.792,A -85,B 0,C 180,E1 -5528.338,E2 -5528.338} C_VEL
LIN {X 0,Y 509.863,Z 253.789,A -85,B 0,C 180,E1 -5531.426,E2 -5531.426} C_VEL
LIN {X 0,Y 509.847,Z 253.79,A -85,B 0,C 180,E1 -5534.67,E2 -5534.67} C_VEL
LIN {X 0,Y 509.841,Z 253.793,A -85,B 0,C 180,E1 -5537.51,E2 -5537.51} C_VEL
LIN {X 0,Y 509.853,Z 253.79,A -85,B 0,C 180,E1 -5540.647,E2 -5540.647} C_VEL
LIN {X 0,Y 509.817,Z 253.796,A -85,B 0,C 180,E1 -5543.645,E2 -5543.645} C_VEL
LIN {X 0,Y 509.867,Z 253.788,A -85,B 0,C 180,E1 -5546.539,E2 -5546.539} C_VEL
LIN {X 0,Y 509.854,Z 253.79,A -85,B 0,C 180,E1 -5549.334,E2 -5549.334} C_VEL
LIN {X 0,Y 509.898,Z 253.784,A -85,B 0,C 180,E1 -5552.054,E2 -5552.054} C_VEL
LIN {X 0,Y 509.849,Z 253.791,A -85,B 0,C 180,E1 -5554.701,E2 -5554.701} C_VEL
LIN {X 0,Y 509.835,Z 253.793,A -85,B 0,C 180,E1 -5557.457,E2 -5557.457} C_VEL
LIN {X 0,Y 509.925,Z 253.78,A -85,B 0,C 180,E1 -5559.844,E2 -5559.844} C_VEL
LIN {X 0,Y 509.88,Z 253.787,A -85,B 0,C 180,E1 -5563.173,E2 -5563.173} C_VEL
LIN {X 0,Y 509.869,Z 253.789,A -85,B 0,C 180,E1 -5565.633,E2 -5565.633} C_VEL
LIN {X 0,Y 509.919,Z 253.784,A -85,B 0,C 180,E1 -5568.873,E2 -5568.873} C_VEL
LIN {X 0,Y 509.928,Z 253.781,A -85,B 0,C 180,E1 -5572.077,E2 -5572.077} C_VEL
LIN {X 0,Y 509.983,Z 253.774,A -85,B 0,C 180,E1 -5574.463,E2 -5574.463} C_VEL
LIN {X 0,Y 510.06,Z 253.764,A -85,B 0,C 180,E1 -5577.63,E2 -5577.63} C_VEL
LIN {X 0,Y 510.069,Z 253.764,A -85,B 0,C 180,E1 -5580.788,E2 -5580.788} C_VEL
LIN {X 0,Y 509.96,Z 253.776,A -85,B 0,C 180,E1 -5583.159,E2 -5583.159} C_VEL
LIN {X 0,Y 509.983,Z 253.774,A -85,B 0,C 180,E1 -5586.328,E2 -5586.328} C_VEL
LIN {X 0,Y 509.918,Z 253.782,A -85,B 0,C 180,E1 -5588.719,E2 -5588.719} C_VEL
LIN {X 0,Y 509.907,Z 253.784,A -85,B 0,C 180,E1 -5591.93,E2 -5591.93} C_VEL
LIN {X 0,Y 509.896,Z 253.785,A -85,B 0,C 180,E1 -5595.24,E2 -5595.24} C_VEL
LIN {X 0,Y 509.89,Z 253.787,A -85,B 0,C 180,E1 -5597.999,E2 -5597.999} C_VEL
LIN {X 0,Y 509.85,Z 253.79,A -85,B 0,C 180,E1 -5601,E2 -5601} C_VEL
LIN {X 0,Y 509.869,Z 253.788,A -85,B 0,C 180,E1 -5604.424,E2 -5604.424} C_VEL
LIN {X 0,Y 509.884,Z 253.785,A -85,B 0,C 180,E1 -5607.054,E2 -5607.054} C_VEL
LIN {X 0,Y 509.854,Z 253.79,A -85,B 0,C 180,E1 -5609.749,E2 -5609.749} C_VEL
LIN {X 0,Y 509.873,Z 253.786,A -85,B 0,C 180,E1 -5612.773,E2 -5612.773} C_VEL
LIN {X 0,Y 509.838,Z 253.793,A -85,B 0,C 180,E1 -5615.579,E2 -5615.579} C_VEL
LIN {X 0,Y 509.845,Z 253.791,A -85,B 0,C 180,E1 -5618.336,E2 -5618.336} C_VEL
LIN {X 0,Y 509.858,Z 253.791,A -85,B 0,C 180,E1 -5621.422,E2 -5621.422} C_VEL
LIN {X 0,Y 509.848,Z 253.791,A -85,B 0,C 180,E1 -5624.666,E2 -5624.666} C_VEL
LIN {X 0,Y 509.877,Z 253.786,A -85,B 0,C 180,E1 -5628.097,E2 -5628.097} C_VEL
LIN {X 0,Y 509.866,Z 253.79,A -85,B 0,C 180,E1 -5630.648,E2 -5630.648} C_VEL
LIN {X 0,Y 509.822,Z 253.793,A -85,B 0,C 180,E1 -5633.721,E2 -5633.721} C_VEL
LIN {X 0,Y 509.155,Z 253.877,A -85,B 0,C 180,E1 -5634.38,E2 -5634.38} C_VEL
LIN {X 0,Y 506.337,Z 254.229,A -85,B 0,C 180,E1 -5635.452,E2 -5635.452} C_VEL
LIN {X 0,Y 503.944,Z 254.528,A -85,B 0,C 180,E1 -5636.316,E2 -5636.316} C_VEL
LIN {X 0,Y 502.895,Z 254.657,A -85,B 0,C 180,E1 -5636.982,E2 -5636.982} C_VEL
LIN {X 0,Y 502.798,Z 254.667,A -85,B 0,C 180,E1 -5637.208,E2 -5637.208} C_VEL
LIN {X 0,Y 502.817,Z 254.666,A -85,B 0,C 180,E1 -5640.06,E2 -5640.06} C_VEL
LIN {X 0,Y 502.821,Z 254.667,A -85,B 0,C 180,E1 -5642.532,E2 -5642.532} C_VEL
LIN {X 0,Y 502.816,Z 254.666,A -85,B 0,C 180,E1 -5645.296,E2 -5645.296} C_VEL
LIN {X 0,Y 502.804,Z 254.668,A -85,B 0,C 180,E1 -5647.827,E2 -5647.827} C_VEL
LIN {X 0,Y 502.796,Z 254.669,A -85,B 0,C 180,E1 -5650.398,E2 -5650.398} C_VEL
LIN {X 0,Y 502.554,Z 254.7,A -85,B 0,C 180,E1 -5652.921,E2 -5652.921} C_VEL
LIN {X 0,Y 502.437,Z 254.722,A -85,B 0,C 180,E1 -5653.753,E2 -5653.753} C_VEL
LIN {X 0,Y 502.427,Z 258.031,A -85,B 0,C 180,E1 -5656.242,E2 -5656.242} C_VEL
LIN {X 0,Y 502.45,Z 261.322,A -85,B 0,C 180,E1 -5658.706,E2 -5658.706} C_VEL
LIN {X 0,Y 502.371,Z 265.693,A -85,B 0,C 180,E1 -5661.957,E2 -5661.957} C_VEL
LIN {X 0,Y 502.436,Z 267.905,A -85,B 0,C 180,E1 -5663.574,E2 -5663.574} C_VEL
LIN {X 0,Y 502.29,Z 272.316,A -85,B 0,C 180,E1 -5666.791,E2 -5666.791} C_VEL
LIN {X 0,Y 502.108,Z 276.766,A -85,B 0,C 180,E1 -5669.999,E2 -5669.999} C_VEL
LIN {X 0,Y 502.158,Z 280.754,A -85,B 0,C 180,E1 -5672.832,E2 -5672.832} C_VEL
LIN {X 0,Y 503.678,Z 290.767,A -85,B 0,C 180,E1 -5673.198,E2 -5673.198} C_VEL
LIN {X 0,Y 503.487,Z 299.726,A -85,B 0,C 180,E1 -5673.6,E2 -5673.6} C_VEL
LIN {X 0,Y 503.302,Z 308.348,A -85,B 0,C 180,E1 -5674.103,E2 -5674.103} C_VEL
LIN {X 0,Y 503.063,Z 316.613,A -85,B 0,C 180,E1 -5674.707,E2 -5674.707} C_VEL
LIN {X 0,Y 502.87,Z 324.427,A -85,B 0,C 180,E1 -5675.412,E2 -5675.412} C_VEL
LIN {X 0,Y 502.711,Z 331.728,A -85,B 0,C 180,E1 -5676.219,E2 -5676.219} C_VEL
LIN {X 0,Y 502.58,Z 339.138,A -85,B 0,C 180,E1 -5677.229,E2 -5677.229} C_VEL
LIN {X 0,Y 502.406,Z 344.975,A -85,B 0,C 180,E1 -5678.243,E2 -5678.243} C_VEL
LIN {X 0,Y 502.256,Z 349.58,A -85,B 0,C 180,E1 -5679.259,E2 -5679.259} C_VEL
LIN {X 0,Y 502.203,Z 352.565,A -85,B 0,C 180,E1 -5680.073,E2 -5680.073} C_VEL
LIN {X 0,Y 502.164,Z 355.789,A -85,B 0,C 180,E1 -5681.298,E2 -5681.298} C_VEL
LIN {X 0,Y 502.083,Z 357.333,A -85,B 0,C 180,E1 -5682.119,E2 -5682.119} C_VEL
LIN {X 0,Y 502.049,Z 358.311,A -85,B 0,C 180,E1 -5682.942,E2 -5682.942} C_VEL
LIN {X 0,Y 502.025,Z 358.703,A -85,B 0,C 180,E1 -5683.767,E2 -5683.767} C_VEL
LIN {X 0,Y 502.072,Z 358.418,A -85,B 0,C 180,E1 -5685.024,E2 -5685.024} C_VEL
LIN {X 0,Y 502.085,Z 356.881,A -85,B 0,C 180,E1 -5686.256,E2 -5686.256} C_VEL
LIN {X 0,Y 502.167,Z 354.063,A -85,B 0,C 180,E1 -5687.5,E2 -5687.5} C_VEL
LIN {X 0,Y 502.292,Z 349.831,A -85,B 0,C 180,E1 -5688.771,E2 -5688.771} C_VEL
LIN {X 0,Y 502.409,Z 344.105,A -85,B 0,C 180,E1 -5690.023,E2 -5690.023} C_VEL
LIN {X 0,Y 502.576,Z 337.497,A -85,B 0,C 180,E1 -5691.104,E2 -5691.104} C_VEL
LIN {X 0,Y 502.761,Z 331.047,A -85,B 0,C 180,E1 -5691.957,E2 -5691.957} C_VEL
LIN {X 0,Y 502.915,Z 323.852,A -85,B 0,C 180,E1 -5692.739,E2 -5692.739} C_VEL
LIN {X 0,Y 503.153,Z 315.753,A -85,B 0,C 180,E1 -5693.457,E2 -5693.457} C_VEL
LIN {X 0,Y 503.443,Z 304.97,A -85,B 0,C 180,E1 -5694.208,E2 -5694.208} C_VEL
LIN {X 0,Y 503.658,Z 295.451,A -85,B 0,C 180,E1 -5694.697,E2 -5694.697} C_VEL
LIN {X 0,Y 503.478,Z 288.478,A -85,B 0,C 180,E1 -5694.989,E2 -5694.989} C_VEL
LIN {X 0,Y 502.13,Z 280.818,A -85,B 0,C 180,E1 -5695.272,E2 -5695.272} C_VEL
LIN {X 0,Y 502.141,Z 276.453,A -85,B 0,C 180,E1 -5698.414,E2 -5698.414} C_VEL
LIN {X 0,Y 502.184,Z 272.356,A -85,B 0,C 180,E1 -5701.39,E2 -5701.39} C_VEL
LIN {X 0,Y 502.21,Z 268.374,A -85,B 0,C 180,E1 -5704.349,E2 -5704.349} C_VEL
LIN {X 0,Y 502.283,Z 264.686,A -85,B 0,C 180,E1 -5707.107,E2 -5707.107} C_VEL
LIN {X 0,Y 502.326,Z 260.809,A -85,B 0,C 180,E1 -5710.058,E2 -5710.058} C_VEL
LIN {X 0,Y 502.47,Z 256.565,A -85,B 0,C 180,E1 -5713.341,E2 -5713.341} C_VEL
LIN {X 0,Y 502.504,Z 255.069,A -85,B 0,C 180,E1 -5714.501,E2 -5714.501} C_VEL
LIN {X 0,Y 502.576,Z 254.697,A -85,B 0,C 180,E1 -5715.641,E2 -5715.641} C_VEL
LIN {X 0,Y 502.772,Z 254.673,A -85,B 0,C 180,E1 -5717.861,E2 -5717.861} C_VEL
LIN {X 0,Y 502.801,Z 254.67,A -85,B 0,C 180,E1 -5721.027,E2 -5721.027} C_VEL
LIN {X 0,Y 502.767,Z 254.675,A -85,B 0,C 180,E1 -5724.168,E2 -5724.168} C_VEL
LIN {X 0,Y 502.813,Z 254.665,A -85,B 0,C 180,E1 -5726.994,E2 -5726.994} C_VEL
LIN {X 0,Y 502.795,Z 254.666,A -85,B 0,C 180,E1 -5730.066,E2 -5730.066} C_VEL
LIN {X 0,Y 502.816,Z 254.665,A -85,B 0,C 180,E1 -5732.534,E2 -5732.534} C_VEL
LIN {X 0,Y 502.808,Z 254.669,A -85,B 0,C 180,E1 -5735.3,E2 -5735.3} C_VEL
LIN {X 0,Y 502.763,Z 254.67,A -85,B 0,C 180,E1 -5737.828,E2 -5737.828} C_VEL
LIN {X 0,Y 502.81,Z 254.666,A -85,B 0,C 180,E1 -5740.402,E2 -5740.402} C_VEL
LIN {X 0,Y 502.819,Z 254.663,A -85,B 0,C 180,E1 -5742.933,E2 -5742.933} C_VEL
LIN {X 0,Y 502.828,Z 254.66,A -85,B 0,C 180,E1 -5745.43,E2 -5745.43} C_VEL
LIN {X 0,Y 502.881,Z 254.654,A -85,B 0,C 180,E1 -5748.719,E2 -5748.719} C_VEL
LIN {X 0,Y 502.887,Z 254.654,A -85,B 0,C 180,E1 -5751.968,E2 -5751.968} C_VEL
LIN {X 0,Y 502.859,Z 254.657,A -85,B 0,C 180,E1 -5755.191,E2 -5755.191} C_VEL
LIN {X 0,Y 503.015,Z 254.641,A -85,B 0,C 180,E1 -5757.599,E2 -5757.599} C_VEL
LIN {X 0,Y 503.013,Z 254.639,A -85,B 0,C 180,E1 -5760.001,E2 -5760.001} C_VEL
LIN {X 0,Y 503.011,Z 254.642,A -85,B 0,C 180,E1 -5762.404,E2 -5762.404} C_VEL
LIN {X 0,Y 502.93,Z 254.65,A -85,B 0,C 180,E1 -5765.615,E2 -5765.615} C_VEL
LIN {X 0,Y 502.89,Z 254.654,A -85,B 0,C 180,E1 -5768.035,E2 -5768.035} C_VEL
LIN {X 0,Y 502.881,Z 254.656,A -85,B 0,C 180,E1 -5771.284,E2 -5771.284} C_VEL
LIN {X 0,Y 502.836,Z 254.662,A -85,B 0,C 180,E1 -5774.572,E2 -5774.572} C_VEL
LIN {X 0,Y 502.807,Z 254.665,A -85,B 0,C 180,E1 -5777.07,E2 -5777.07} C_VEL
LIN {X 0,Y 502.811,Z 254.668,A -85,B 0,C 180,E1 -5779.601,E2 -5779.601} C_VEL
LIN {X 0,Y 502.791,Z 254.67,A -85,B 0,C 180,E1 -5782.703,E2 -5782.703} C_VEL
LIN {X 0,Y 502.803,Z 254.667,A -85,B 0,C 180,E1 -5785.679,E2 -5785.679} C_VEL
LIN {X 0,Y 502.789,Z 254.668,A -85,B 0,C 180,E1 -5788.377,E2 -5788.377} C_VEL
LIN {X 0,Y 502.791,Z 254.67,A -85,B 0,C 180,E1 -5791.145,E2 -5791.145} C_VEL
LIN {X 0,Y 502.797,Z 254.672,A -85,B 0,C 180,E1 -5793.995,E2 -5793.995} C_VEL
LIN {X 0,Y 502.759,Z 254.676,A -85,B 0,C 180,E1 -5797.177,E2 -5797.177} C_VEL
LIN {X 0,Y 502.816,Z 254.666,A -85,B 0,C 180,E1 -5800.013,E2 -5800.013} C_VEL
LIN {X 0,Y 502.767,Z 254.673,A -85,B 0,C 180,E1 -5803.233,E2 -5803.233} C_VEL
LIN {X 0,Y 502.774,Z 254.67,A -85,B 0,C 180,E1 -5805.661,E2 -5805.661} C_VEL
LIN {X 0,Y 502.816,Z 254.665,A -85,B 0,C 180,E1 -5809.006,E2 -5809.006} C_VEL
LIN {X 0,Y 502.788,Z 254.671,A -85,B 0,C 180,E1 -5812.047,E2 -5812.047} C_VEL
LIN {X 0,Y 502.801,Z 254.698,A -85,B 0,C 180,E1 -5814.453,E2 -5814.453} C_VEL
LIN {X 0,Y 503.763,Z 260.268,A -85,B 0,C 180,E1 -5816.832,E2 -5816.832} C_VEL
LIN {X 0,Y 503.65,Z 265.581,A -85,B 0,C 180,E1 -5818.917,E2 -5818.917} C_VEL
LIN {X 0,Y 503.334,Z 272.876,A -85,B 0,C 180,E1 -5821.659,E2 -5821.659} C_VEL
LIN {X 0,Y 503.012,Z 281.53,A -85,B 0,C 180,E1 -5824.779,E2 -5824.779} C_VEL
LIN {X 0,Y 502.752,Z 290.301,A -85,B 0,C 180,E1 -5827.826,E2 -5827.826} C_VEL
LIN {X 0,Y 502.533,Z 299.133,A -85,B 0,C 180,E1 -5830.814,E2 -5830.814} C_VEL
LIN {X 0,Y 502.431,Z 308.034,A -85,B 0,C 180,E1 -5833.755,E2 -5833.755} C_VEL
LIN {X 0,Y 502.267,Z 316.987,A -85,B 0,C 180,E1 -5836.652,E2 -5836.652} C_VEL
LIN {X 0,Y 502.292,Z 323.36,A -85,B 0,C 180,E1 -5838.705,E2 -5838.705} C_VEL
LIN {X 0,Y 503.534,Z 336.485,A -85,B 0,C 180,E1 -5839.14,E2 -5839.14} C_VEL
LIN {X 0,Y 503.361,Z 345.559,A -85,B 0,C 180,E1 -5839.544,E2 -5839.544} C_VEL
LIN {X 0,Y 503.186,Z 354.297,A -85,B 0,C 180,E1 -5840.048,E2 -5840.048} C_VEL
LIN {X 0,Y 502.964,Z 362.643,A -85,B 0,C 180,E1 -5840.653,E2 -5840.653} C_VEL
LIN {X 0,Y 502.741,Z 370.545,A -85,B 0,C 180,E1 -5841.358,E2 -5841.358} C_VEL
LIN {X 0,Y 502.544,Z 377.936,A -85,B 0,C 180,E1 -5842.164,E2 -5842.164} C_VEL
LIN {X 0,Y 502.363,Z 385.443,A -85,B 0,C 180,E1 -5843.172,E2 -5843.172} C_VEL
LIN {X 0,Y 502.267,Z 392.298,A -85,B 0,C 180,E1 -5844.38,E2 -5844.38} C_VEL
LIN {X 0,Y 502.134,Z 397.502,A -85,B 0,C 180,E1 -5845.586,E2 -5845.586} C_VEL
LIN {X 0,Y 502.164,Z 400.168,A -85,B 0,C 180,E1 -5846.39,E2 -5846.39} C_VEL
LIN {X 0,Y 502.123,Z 403.089,A -85,B 0,C 180,E1 -5847.595,E2 -5847.595} C_VEL
LIN {X 0,Y 502.035,Z 404.347,A -85,B 0,C 180,E1 -5848.397,E2 -5848.397} C_VEL
LIN {X 0,Y 501.99,Z 405.132,A -85,B 0,C 180,E1 -5849.199,E2 -5849.199} C_VEL
LIN {X 0,Y 501.986,Z 405.43,A -85,B 0,C 180,E1 -5850.001,E2 -5850.001} C_VEL
LIN {X 0,Y 501.99,Z 405.135,A -85,B 0,C 180,E1 -5850.803,E2 -5850.803} C_VEL
LIN {X 0,Y 502.036,Z 404.353,A -85,B 0,C 180,E1 -5851.605,E2 -5851.605} C_VEL
LIN {X 0,Y 502.123,Z 403.096,A -85,B 0,C 180,E1 -5852.408,E2 -5852.408} C_VEL
LIN {X 0,Y 502.164,Z 400.18,A -85,B 0,C 180,E1 -5853.612,E2 -5853.612} C_VEL
LIN {X 0,Y 502.134,Z 397.517,A -85,B 0,C 180,E1 -5854.416,E2 -5854.416} C_VEL
LIN {X 0,Y 502.268,Z 392.315,A -85,B 0,C 180,E1 -5855.622,E2 -5855.622} C_VEL
LIN {X 0,Y 502.414,Z 385.461,A -85,B 0,C 180,E1 -5856.829,E2 -5856.829} C_VEL
LIN {X 0,Y 502.549,Z 377.965,A -85,B 0,C 180,E1 -5857.838,E2 -5857.838} C_VEL
LIN {X 0,Y 502.743,Z 370.579,A -85,B 0,C 180,E1 -5858.644,E2 -5858.644} C_VEL
LIN {X 0,Y 502.964,Z 362.674,A -85,B 0,C 180,E1 -5859.349,E2 -5859.349} C_VEL
LIN {X 0,Y 503.142,Z 354.323,A -85,B 0,C 180,E1 -5859.955,E2 -5859.955} C_VEL
LIN {X 0,Y 503.446,Z 343.669,A -85,B 0,C 180,E1 -5860.558,E2 -5860.558} C_VEL
LIN {X 0,Y 503.475,Z 335.247,A -85,B 0,C 180,E1 -5860.914,E2 -5860.914} C_VEL
LIN {X 0,Y 502.247,Z 323.424,A -85,B 0,C 180,E1 -5861.298,E2 -5861.298} C_VEL
LIN {X 0,Y 502.346,Z 313.253,A -85,B 0,C 180,E1 -5864.587,E2 -5864.587} C_VEL
LIN {X 0,Y 502.464,Z 304.326,A -85,B 0,C 180,E1 -5867.502,E2 -5867.502} C_VEL
LIN {X 0,Y 502.669,Z 294.14,A -85,B 0,C 180,E1 -5870.887,E2 -5870.887} C_VEL
LIN {X 0,Y 502.882,Z 285.247,A -85,B 0,C 180,E1 -5873.91,E2 -5873.91} C_VEL
LIN {X 0,Y 503.183,Z 276.381,A -85,B 0,C 180,E1 -5876.997,E2 -5876.997} C_VEL
LIN {X 0,Y 503.48,Z 267.559,A -85,B 0,C 180,E1 -5880.168,E2 -5880.168} C_VEL
LIN {X 0,Y 503.671,Z 261.281,A -85,B 0,C 180,E1 -5882.495,E2 -5882.495} C_VEL
LIN {X 0,Y 503.335,Z 257.535,A -85,B 0,C 180,E1 -5883.954,E2 -5883.954} C_VEL
LIN {X 0,Y 502.802,Z 254.67,A -85,B 0,C 180,E1 -5885.15,E2 -5885.15} C_VEL
LIN {X 0,Y 502.802,Z 254.669,A -85,B 0,C 180,E1 -5888.486,E2 -5888.486} C_VEL
LIN {X 0,Y 502.827,Z 254.664,A -85,B 0,C 180,E1 -5891.066,E2 -5891.066} C_VEL
LIN {X 0,Y 502.794,Z 254.669,A -85,B 0,C 180,E1 -5894.53,E2 -5894.53} C_VEL
LIN {X 0,Y 502.803,Z 254.669,A -85,B 0,C 180,E1 -5897.861,E2 -5897.861} C_VEL
LIN {X 0,Y 502.808,Z 254.666,A -85,B 0,C 180,E1 -5901.024,E2 -5901.024} C_VEL
LIN {X 0,Y 502.779,Z 254.671,A -85,B 0,C 180,E1 -5904.169,E2 -5904.169} C_VEL
LIN {X 0,Y 502.841,Z 254.663,A -85,B 0,C 180,E1 -5906.993,E2 -5906.993} C_VEL
LIN {X 0,Y 502.824,Z 254.665,A -85,B 0,C 180,E1 -5910.065,E2 -5910.065} C_VEL
LIN {X 0,Y 502.839,Z 254.663,A -85,B 0,C 180,E1 -5912.533,E2 -5912.533} C_VEL
LIN {X 0,Y 502.812,Z 254.667,A -85,B 0,C 180,E1 -5915.304,E2 -5915.304} C_VEL
LIN {X 0,Y 502.788,Z 254.67,A -85,B 0,C 180,E1 -5917.826,E2 -5917.826} C_VEL
LIN {X 0,Y 502.832,Z 254.663,A -85,B 0,C 180,E1 -5920.399,E2 -5920.399} C_VEL
LIN {X 0,Y 502.826,Z 254.666,A -85,B 0,C 180,E1 -5922.93,E2 -5922.93} C_VEL
LIN {X 0,Y 502.851,Z 254.663,A -85,B 0,C 180,E1 -5925.428,E2 -5925.428} C_VEL
LIN {X 0,Y 502.884,Z 254.659,A -85,B 0,C 180,E1 -5928.716,E2 -5928.716} C_VEL
LIN {X 0,Y 502.887,Z 254.658,A -85,B 0,C 180,E1 -5931.965,E2 -5931.965} C_VEL
LIN {X 0,Y 502.937,Z 254.651,A -85,B 0,C 180,E1 -5934.385,E2 -5934.385} C_VEL
LIN {X 0,Y 503.03,Z 254.639,A -85,B 0,C 180,E1 -5937.596,E2 -5937.596} C_VEL
LIN {X 0,Y 503.033,Z 254.64,A -85,B 0,C 180,E1 -5939.999,E2 -5939.999} C_VEL
LIN {X 0,Y 503.03,Z 254.64,A -85,B 0,C 180,E1 -5942.401,E2 -5942.401} C_VEL
LIN {X 0,Y 502.933,Z 254.652,A -85,B 0,C 180,E1 -5946.417,E2 -5946.417} C_VEL
LIN {X 0,Y 502.877,Z 254.66,A -85,B 0,C 180,E1 -5948.842,E2 -5948.842} C_VEL
LIN {X 0,Y 502.849,Z 254.664,A -85,B 0,C 180,E1 -5952.1,E2 -5952.1} C_VEL
LIN {X 0,Y 502.85,Z 254.662,A -85,B 0,C 180,E1 -5955.398,E2 -5955.398} C_VEL
LIN {X 0,Y 502.847,Z 254.665,A -85,B 0,C 180,E1 -5958.12,E2 -5958.12} C_VEL
LIN {X 0,Y 502.829,Z 254.664,A -85,B 0,C 180,E1 -5960.534,E2 -5960.534} C_VEL
LIN {X 0,Y 502.794,Z 254.669,A -85,B 0,C 180,E1 -5963.038,E2 -5963.038} C_VEL
LIN {X 0,Y 502.839,Z 254.664,A -85,B 0,C 180,E1 -5965.673,E2 -5965.673} C_VEL
LIN {X 0,Y 502.838,Z 254.663,A -85,B 0,C 180,E1 -5968.371,E2 -5968.371} C_VEL
LIN {X 0,Y 502.793,Z 254.671,A -85,B 0,C 180,E1 -5971.497,E2 -5971.497} C_VEL
LIN {X 0,Y 502.802,Z 254.668,A -85,B 0,C 180,E1 -5974.443,E2 -5974.443} C_VEL
LIN {X 0,Y 502.775,Z 254.672,A -85,B 0,C 180,E1 -5977.176,E2 -5977.176} C_VEL
LIN {X 0,Y 502.815,Z 254.667,A -85,B 0,C 180,E1 -5980.01,E2 -5980.01} C_VEL
LIN {X 0,Y 502.822,Z 254.666,A -85,B 0,C 180,E1 -5982.201,E2 -5982.201} C_VEL
LIN {X 0,Y 502.792,Z 254.671,A -85,B 0,C 180,E1 -5985.466,E2 -5985.466} C_VEL
LIN {X 0,Y 502.829,Z 254.664,A -85,B 0,C 180,E1 -5987.863,E2 -5987.863} C_VEL
LIN {X 0,Y 502.811,Z 254.667,A -85,B 0,C 180,E1 -5991.024,E2 -5991.024} C_VEL
LIN {X 0,Y 502.775,Z 254.67,A -85,B 0,C 180,E1 -5994.165,E2 -5994.165} C_VEL
LIN {X 0,Y 502.798,Z 254.667,A -85,B 0,C 180,E1 -5997.208,E2 -5997.208} C_VEL
LIN {X 0,Y 502.099,Z 254.755,A -85,B 0,C 180,E1 -5997.876,E2 -5997.876} C_VEL
LIN {X 0,Y 499.241,Z 255.112,A -85,B 0,C 180,E1 -5998.962,E2 -5998.962} C_VEL
LIN {X 0,Y 496.849,Z 255.409,A -85,B 0,C 180,E1 -5999.837,E2 -5999.837} C_VEL
LIN {X 0,Y 495.83,Z 255.537,A -85,B 0,C 180,E1 -6000.513,E2 -6000.513} C_VEL
LIN {X 0,Y 495.751,Z 255.544,A -85,B 0,C 180,E1 -6000.741,E2 -6000.741} C_VEL
LIN {X 0,Y 495.785,Z 255.542,A -85,B 0,C 180,E1 -6003.931,E2 -6003.931} C_VEL
LIN {X 0,Y 495.771,Z 255.544,A -85,B 0,C 180,E1 -6007.13,E2 -6007.13} C_VEL
LIN {X 0,Y 495.753,Z 255.547,A -85,B 0,C 180,E1 -6010.108,E2 -6010.108} C_VEL
LIN {X 0,Y 495.695,Z 255.554,A -85,B 0,C 180,E1 -6011.824,E2 -6011.824} C_VEL
LIN {X 0,Y 495.423,Z 255.588,A -85,B 0,C 180,E1 -6013.517,E2 -6013.517} C_VEL
LIN {X 0,Y 495.456,Z 256.659,A -85,B 0,C 180,E1 -6014.693,E2 -6014.693} C_VEL
LIN {X 0,Y 495.461,Z 261.235,A -85,B 0,C 180,E1 -6018.154,E2 -6018.154} C_VEL
LIN {X 0,Y 495.301,Z 266.173,A -85,B 0,C 180,E1 -6021.842,E2 -6021.842} C_VEL
LIN {X 0,Y 495.376,Z 268.375,A -85,B 0,C 180,E1 -6023.482,E2 -6023.482} C_VEL
LIN {X 0,Y 495.236,Z 272.827,A -85,B 0,C 180,E1 -6026.745,E2 -6026.745} C_VEL
LIN {X 0,Y 495.029,Z 277.325,A -85,B 0,C 180,E1 -6029.999,E2 -6029.999} C_VEL
LIN {X 0,Y 495.064,Z 281.033,A -85,B 0,C 180,E1 -6032.669,E2 -6032.669} C_VEL
LIN {X 0,Y 496.699,Z 290.983,A -85,B 0,C 180,E1 -6033.04,E2 -6033.04} C_VEL
LIN {X 0,Y 496.532,Z 299.949,A -85,B 0,C 180,E1 -6033.448,E2 -6033.448} C_VEL
LIN {X 0,Y 496.33,Z 308.596,A -85,B 0,C 180,E1 -6033.957,E2 -6033.957} C_VEL
LIN {X 0,Y 496.067,Z 316.881,A -85,B 0,C 180,E1 -6034.57,E2 -6034.57} C_VEL
LIN {X 0,Y 495.858,Z 324.708,A -85,B 0,C 180,E1 -6035.285,E2 -6035.285} C_VEL
LIN {X 0,Y 495.681,Z 332.018,A -85,B 0,C 180,E1 -6036.103,E2 -6036.103} C_VEL
LIN {X 0,Y 495.552,Z 339.5,A -85,B 0,C 180,E1 -6037.138,E2 -6037.138} C_VEL
LIN {X 0,Y 495.34,Z 345.282,A -85,B 0,C 180,E1 -6038.156,E2 -6038.156} C_VEL
LIN {X 0,Y 495.209,Z 349.101,A -85,B 0,C 180,E1 -6038.98,E2 -6038.98} C_VEL
LIN {X 0,Y 495.136,Z 353.462,A -85,B 0,C 180,E1 -6040.219,E2 -6040.219} C_VEL
LIN {X 0,Y 495.06,Z 356.837,A -85,B 0,C 180,E1 -6041.623,E2 -6041.623} C_VEL
LIN {X 0,Y 494.957,Z 358.781,A -85,B 0,C 180,E1 -6043.13,E2 -6043.13} C_VEL
LIN {X 0,Y 494.961,Z 359.108,A -85,B 0,C 180,E1 -6043.967,E2 -6043.967} C_VEL
LIN {X 0,Y 494.98,Z 358.702,A -85,B 0,C 180,E1 -6045.104,E2 -6045.104} C_VEL
LIN {X 0,Y 495.016,Z 356.803,A -85,B 0,C 180,E1 -6046.495,E2 -6046.495} C_VEL
LIN {X 0,Y 495.095,Z 354.973,A -85,B 0,C 180,E1 -6047.342,E2 -6047.342} C_VEL
LIN {X 0,Y 495.163,Z 352.534,A -85,B 0,C 180,E1 -6048.194,E2 -6048.194} C_VEL
LIN {X 0,Y 495.265,Z 349.382,A -85,B 0,C 180,E1 -6049.048,E2 -6049.048} C_VEL
LIN {X 0,Y 495.41,Z 343.696,A -85,B 0,C 180,E1 -6050.238,E2 -6050.238} C_VEL
LIN {X 0,Y 495.543,Z 337.859,A -85,B 0,C 180,E1 -6051.2,E2 -6051.2} C_VEL
LIN {X 0,Y 495.734,Z 331.415,A -85,B 0,C 180,E1 -6052.066,E2 -6052.066} C_VEL
LIN {X 0,Y 495.9,Z 324.7,A -85,B 0,C 180,E1 -6052.811,E2 -6052.811} C_VEL
LIN {X 0,Y 496.123,Z 317.447,A -85,B 0,C 180,E1 -6053.478,E2 -6053.478} C_VEL
LIN {X 0,Y 496.364,Z 310.315,A -85,B 0,C 180,E1 -6054.02,E2 -6054.02} C_VEL
LIN {X 0,Y 496.559,Z 302.101,A -85,B 0,C 180,E1 -6054.528,E2 -6054.528} C_VEL
LIN {X 0,Y 496.71,Z 293.245,A -85,B 0,C 180,E1 -6054.957,E2 -6054.957} C_VEL
LIN {X 0,Y 496.282,Z 288.109,A -85,B 0,C 180,E1 -6055.173,E2 -6055.173} C_VEL
LIN {X 0,Y 495.046,Z 281.158,A -85,B 0,C 180,E1 -6055.431,E2 -6055.431} C_VEL
LIN {X 0,Y 495.066,Z 276.418,A -85,B 0,C 180,E1 -6058.858,E2 -6058.858} C_VEL
LIN {X 0,Y 495.118,Z 272.586,A -85,B 0,C 180,E1 -6061.68,E2 -6061.68} C_VEL
LIN {X 0,Y 495.138,Z 268.693,A -85,B 0,C 180,E1 -6064.593,E2 -6064.593} C_VEL
LIN {X 0,Y 495.217,Z 264.749,A -85,B 0,C 180,E1 -6067.605,E2 -6067.605} C_VEL
LIN {X 0,Y 495.309,Z 260.659,A -85,B 0,C 180,E1 -6070.744,E2 -6070.744} C_VEL
LIN {X 0,Y 495.433,Z 256.456,A -85,B 0,C 180,E1 -6074.033,E2 -6074.033} C_VEL
LIN {X 0,Y 495.443,Z 255.587,A -85,B 0,C 180,E1 -6074.828,E2 -6074.828} C_VEL
LIN {X 0,Y 495.701,Z 255.55,A -85,B 0,C 180,E1 -6077.496,E2 -6077.496} C_VEL
LIN {X 0,Y 495.771,Z 255.541,A -85,B 0,C 180,E1 -6080.366,E2 -6080.366} C_VEL
LIN {X 0,Y 495.716,Z 255.549,A -85,B 0,C 180,E1 -6083.458,E2 -6083.458} C_VEL
LIN {X 0,Y 495.741,Z 255.545,A -85,B 0,C 180,E1 -6086.437,E2 -6086.437} C_VEL
LIN {X 0,Y 495.732,Z 255.548,A -85,B 0,C 180,E1 -6089.314,E2 -6089.314} C_VEL
LIN {X 0,Y 495.764,Z 255.546,A -85,B 0,C 180,E1 -6092.11,E2 -6092.11} C_VEL
LIN {X 0,Y 495.754,Z 255.544,A -85,B 0,C 180,E1 -6094.833,E2 -6094.833} C_VEL
LIN {X 0,Y 495.731,Z 255.546,A -85,B 0,C 180,E1 -6097.496,E2 -6097.496} C_VEL
LIN {X 0,Y 495.763,Z 255.546,A -85,B 0,C 180,E1 -6100.111,E2 -6100.111} C_VEL
LIN {X 0,Y 495.771,Z 255.539,A -85,B 0,C 180,E1 -6102.683,E2 -6102.683} C_VEL
LIN {X 0,Y 495.773,Z 255.54,A -85,B 0,C 180,E1 -6105.218,E2 -6105.218} C_VEL
LIN {X 0,Y 495.856,Z 255.53,A -85,B 0,C 180,E1 -6108.557,E2 -6108.557} C_VEL
LIN {X 0,Y 495.858,Z 255.53,A -85,B 0,C 180,E1 -6111.853,E2 -6111.853} C_VEL
LIN {X 0,Y 495.827,Z 255.533,A -85,B 0,C 180,E1 -6115.123,E2 -6115.123} C_VEL
LIN {X 0,Y 495.984,Z 255.517,A -85,B 0,C 180,E1 -6117.565,E2 -6117.565} C_VEL
LIN {X 0,Y 495.984,Z 255.514,A -85,B 0,C 180,E1 -6120.001,E2 -6120.001} C_VEL
LIN {X 0,Y 495.98,Z 255.518,A -85,B 0,C 180,E1 -6122.438,E2 -6122.438} C_VEL
LIN {X 0,Y 495.887,Z 255.527,A -85,B 0,C 180,E1 -6125.695,E2 -6125.695} C_VEL
LIN {X 0,Y 495.861,Z 255.531,A -85,B 0,C 180,E1 -6128.149,E2 -6128.149} C_VEL
LIN {X 0,Y 495.867,Z 255.531,A -85,B 0,C 180,E1 -6132.062,E2 -6132.062} C_VEL
LIN {X 0,Y 495.798,Z 255.538,A -85,B 0,C 180,E1 -6135.625,E2 -6135.625} C_VEL
LIN {X 0,Y 495.77,Z 255.541,A -85,B 0,C 180,E1 -6139.03,E2 -6139.03} C_VEL
LIN {X 0,Y 495.739,Z 255.547,A -85,B 0,C 180,E1 -6141.63,E2 -6141.63} C_VEL
LIN {X 0,Y 495.763,Z 255.544,A -85,B 0,C 180,E1 -6144.873,E2 -6144.873} C_VEL
LIN {X 0,Y 495.734,Z 255.549,A -85,B 0,C 180,E1 -6147.895,E2 -6147.895} C_VEL
LIN {X 0,Y 495.746,Z 255.55,A -85,B 0,C 180,E1 -6150.689,E2 -6150.689} C_VEL
LIN {X 0,Y 495.753,Z 255.547,A -85,B 0,C 180,E1 -6153.566,E2 -6153.566} C_VEL
LIN {X 0,Y 495.71,Z 255.55,A -85,B 0,C 180,E1 -6156.546,E2 -6156.546} C_VEL
LIN {X 0,Y 495.778,Z 255.541,A -85,B 0,C 180,E1 -6159.637,E2 -6159.637} C_VEL
LIN {X 0,Y 495.732,Z 255.547,A -85,B 0,C 180,E1 -6162.508,E2 -6162.508} C_VEL
LIN {X 0,Y 495.732,Z 255.551,A -85,B 0,C 180,E1 -6165.142,E2 -6165.142} C_VEL
LIN {X 0,Y 495.754,Z 255.549,A -85,B 0,C 180,E1 -6168.22,E2 -6168.22} C_VEL
LIN {X 0,Y 495.746,Z 255.55,A -85,B 0,C 180,E1 -6171.41,E2 -6171.41} C_VEL
LIN {X 0,Y 495.762,Z 255.688,A -85,B 0,C 180,E1 -6174.263,E2 -6174.263} C_VEL
LIN {X 0,Y 496.71,Z 261.04,A -85,B 0,C 180,E1 -6176.595,E2 -6176.595} C_VEL
LIN {X 0,Y 496.734,Z 265.592,A -85,B 0,C 180,E1 -6178.435,E2 -6178.435} C_VEL
LIN {X 0,Y 496.318,Z 274.241,A -85,B 0,C 180,E1 -6181.764,E2 -6181.764} C_VEL
LIN {X 0,Y 495.926,Z 283.367,A -85,B 0,C 180,E1 -6185.091,E2 -6185.091} C_VEL
LIN {X 0,Y 495.69,Z 291.387,A -85,B 0,C 180,E1 -6187.932,E2 -6187.932} C_VEL
LIN {X 0,Y 495.457,Z 300.222,A -85,B 0,C 180,E1 -6190.96,E2 -6190.96} C_VEL
LIN {X 0,Y 495.353,Z 309.063,A -85,B 0,C 180,E1 -6193.94,E2 -6193.94} C_VEL
LIN {X 0,Y 495.174,Z 317.966,A -85,B 0,C 180,E1 -6196.876,E2 -6196.876} C_VEL
LIN {X 0,Y 495.218,Z 323.348,A -85,B 0,C 180,E1 -6198.567,E2 -6198.567} C_VEL
LIN {X 0,Y 496.408,Z 334.887,A -85,B 0,C 180,E1 -6198.931,E2 -6198.931} C_VEL
LIN {X 0,Y 496.362,Z 345.217,A -85,B 0,C 180,E1 -6199.394,E2 -6199.394} C_VEL
LIN {X 0,Y 496.181,Z 353.956,A -85,B 0,C 180,E1 -6199.906,E2 -6199.906} C_VEL
LIN {X 0,Y 495.949,Z 362.303,A -85,B 0,C 180,E1 -6200.519,E2 -6200.519} C_VEL
LIN {X 0,Y 495.698,Z 370.205,A -85,B 0,C 180,E1 -6201.234,E2 -6201.234} C_VEL
LIN {X 0,Y 495.471,Z 377.597,A -85,B 0,C 180,E1 -6202.052,E2 -6202.052} C_VEL
LIN {X 0,Y 495.298,Z 385.106,A -85,B 0,C 180,E1 -6203.074,E2 -6203.074} C_VEL
LIN {X 0,Y 495.198,Z 391.963,A -85,B 0,C 180,E1 -6204.3,E2 -6204.3} C_VEL
LIN {X 0,Y 495.039,Z 397.168,A -85,B 0,C 180,E1 -6205.523,E2 -6205.523} C_VEL
LIN {X 0,Y 495.058,Z 400.997,A -85,B 0,C 180,E1 -6206.746,E2 -6206.746} C_VEL
LIN {X 0,Y 495.027,Z 402.758,A -85,B 0,C 180,E1 -6207.56,E2 -6207.56} C_VEL
LIN {X 0,Y 494.962,Z 404.017,A -85,B 0,C 180,E1 -6208.374,E2 -6208.374} C_VEL
LIN {X 0,Y 494.91,Z 404.802,A -85,B 0,C 180,E1 -6209.187,E2 -6209.187} C_VEL
LIN {X 0,Y 494.903,Z 405.101,A -85,B 0,C 180,E1 -6210.001,E2 -6210.001} C_VEL
LIN {X 0,Y 494.91,Z 404.807,A -85,B 0,C 180,E1 -6210.815,E2 -6210.815} C_VEL
LIN {X 0,Y 494.963,Z 404.024,A -85,B 0,C 180,E1 -6211.628,E2 -6211.628} C_VEL
LIN {X 0,Y 495.027,Z 402.767,A -85,B 0,C 180,E1 -6212.442,E2 -6212.442} C_VEL
LIN {X 0,Y 495.085,Z 399.851,A -85,B 0,C 180,E1 -6213.664,E2 -6213.664} C_VEL
LIN {X 0,Y 495.039,Z 397.187,A -85,B 0,C 180,E1 -6214.479,E2 -6214.479} C_VEL
LIN {X 0,Y 495.199,Z 391.986,A -85,B 0,C 180,E1 -6215.703,E2 -6215.703} C_VEL
LIN {X 0,Y 495.34,Z 385.131,A -85,B 0,C 180,E1 -6216.927,E2 -6216.927} C_VEL
LIN {X 0,Y 495.476,Z 377.633,A -85,B 0,C 180,E1 -6217.95,E2 -6217.95} C_VEL
LIN {X 0,Y 495.7,Z 370.248,A -85,B 0,C 180,E1 -6218.768,E2 -6218.768} C_VEL
LIN {X 0,Y 495.951,Z 362.344,A -85,B 0,C 180,E1 -6219.483,E2 -6219.483} C_VEL
LIN {X 0,Y 496.139,Z 353.992,A -85,B 0,C 180,E1 -6220.097,E2 -6220.097} C_VEL
LIN {X 0,Y 496.458,Z 343.338,A -85,B 0,C 180,E1 -6220.709,E2 -6220.709} C_VEL
LIN {X 0,Y 496.384,Z 334.91,A -85,B 0,C 180,E1 -6221.072,E2 -6221.072} C_VEL
LIN {X 0,Y 495.156,Z 323.14,A -85,B 0,C 180,E1 -6221.462,E2 -6221.462} C_VEL
LIN {X 0,Y 495.27,Z 312.98,A -85,B 0,C 180,E1 -6224.8,E2 -6224.8} C_VEL
LIN {X 0,Y 495.384,Z 304.191,A -85,B 0,C 180,E1 -6227.721,E2 -6227.721} C_VEL
LIN {X 0,Y 495.59,Z 295.173,A -85,B 0,C 180,E1 -6230.765,E2 -6230.765} C_VEL
LIN {X 0,Y 495.822,Z 286.296,A -85,B 0,C 180,E1 -6233.828,E2 -6233.828} C_VEL
LIN {X 0,Y 496.127,Z 277.442,A -85,B 0,C 180,E1 -6236.957,E2 -6236.957} C_VEL
LIN {X 0,Y 496.428,Z 269.883,A -85,B 0,C 180,E1 -6239.704,E2 -6239.704} C_VEL
LIN {X 0,Y 496.671,Z 262.36,A -85,B 0,C 180,E1 -6242.529,E2 -6242.529} C_VEL
LIN {X 0,Y 496.333,Z 258.617,A -85,B 0,C 180,E1 -6244.009,E2 -6244.009} C_VEL
LIN {X 0,Y 495.77,Z 255.546,A -85,B 0,C 180,E1 -6245.318,E2 -6245.318} C_VEL
LIN {X 0,Y 495.77,Z 255.544,A -85,B 0,C 180,E1 -6248.768,E2 -6248.768} C_VEL
LIN {X 0,Y 495.764,Z 255.545,A -85,B 0,C 180,E1 -6251.781,E2 -6251.781} C_VEL
LIN {X 0,Y 495.745,Z 255.546,A -85,B 0,C 180,E1 -6255.141,E2 -6255.141} C_VEL
LIN {X 0,Y 495.764,Z 255.546,A -85,B 0,C 180,E1 -6258.219,E2 -6258.219} C_VEL
LIN {X 0,Y 495.757,Z 255.546,A -85,B 0,C 180,E1 -6261.408,E2 -6261.408} C_VEL
LIN {X 0,Y 495.753,Z 255.546,A -85,B 0,C 180,E1 -6264.462,E2 -6264.462} C_VEL
LIN {X 0,Y 495.776,Z 255.544,A -85,B 0,C 180,E1 -6267.405,E2 -6267.405} C_VEL
LIN {X 0,Y 495.775,Z 255.543,A -85,B 0,C 180,E1 -6270.253,E2 -6270.253} C_VEL
LIN {X 0,Y 495.832,Z 255.537,A -85,B 0,C 180,E1 -6273.25,E2 -6273.25} C_VEL
LIN {X 0,Y 495.751,Z 255.546,A -85,B 0,C 180,E1 -6276.612,E2 -6276.612} C_VEL
LIN {X 0,Y 495.787,Z 255.543,A -85,B 0,C 180,E1 -6279.323,E2 -6279.323} C_VEL
LIN {X 0,Y 495.789,Z 255.541,A -85,B 0,C 180,E1 -6281.828,E2 -6281.828} C_VEL
LIN {X 0,Y 495.832,Z 255.536,A -85,B 0,C 180,E1 -6284.548,E2 -6284.548} C_VEL
LIN {X 0,Y 495.836,Z 255.535,A -85,B 0,C 180,E1 -6287.964,E2 -6287.964} C_VEL
LIN {X 0,Y 495.841,Z 255.536,A -85,B 0,C 180,E1 -6291.029,E2 -6291.029} C_VEL
LIN {X 0,Y 495.866,Z 255.532,A -85,B 0,C 180,E1 -6293.488,E2 -6293.488} C_VEL
LIN {X 0,Y 495.847,Z 255.536,A -85,B 0,C 180,E1 -6296.748,E2 -6296.748} C_VEL
LIN {X 0,Y 495.875,Z 255.531,A -85,B 0,C 180,E1 -6298.374,E2 -6298.374} C_VEL
LIN {X 0,Y 496.01,Z 255.516,A -85,B 0,C 180,E1 -6300.81,E2 -6300.81} C_VEL
LIN {X 0,Y 495.847,Z 255.533,A -85,B 0,C 180,E1 -6303.249,E2 -6303.249} C_VEL
LIN {X 0,Y 495.884,Z 255.53,A -85,B 0,C 180,E1 -6306.509,E2 -6306.509} C_VEL
LIN {X 0,Y 495.846,Z 255.535,A -85,B 0,C 180,E1 -6308.968,E2 -6308.968} C_VEL
LIN {X 0,Y 495.831,Z 255.538,A -85,B 0,C 180,E1 -6312.033,E2 -6312.033} C_VEL
LIN {X 0,Y 495.826,Z 255.537,A -85,B 0,C 180,E1 -6315.45,E2 -6315.45} C_VEL
LIN {X 0,Y 495.808,Z 255.54,A -85,B 0,C 180,E1 -6318.245,E2 -6318.245} C_VEL
LIN {X 0,Y 495.774,Z 255.543,A -85,B 0,C 180,E1 -6320.754,E2 -6320.754} C_VEL
LIN {X 0,Y 495.751,Z 255.548,A -85,B 0,C 180,E1 -6323.385,E2 -6323.385} C_VEL
LIN {X 0,Y 495.789,Z 255.543,A -85,B 0,C 180,E1 -6326.066,E2 -6326.066} C_VEL
LIN {X 0,Y 495.769,Z 255.542,A -85,B 0,C 180,E1 -6328.813,E2 -6328.813} C_VEL
LIN {X 0,Y 495.755,Z 255.546,A -85,B 0,C 180,E1 -6331.724,E2 -6331.724} C_VEL
LIN {X 0,Y 495.772,Z 255.543,A -85,B 0,C 180,E1 -6334.693,E2 -6334.693} C_VEL
LIN {X 0,Y 495.726,Z 255.551,A -85,B 0,C 180,E1 -6337.559,E2 -6337.559} C_VEL
LIN {X 0,Y 495.773,Z 255.544,A -85,B 0,C 180,E1 -6340.696,E2 -6340.696} C_VEL
LIN {X 0,Y 495.726,Z 255.55,A -85,B 0,C 180,E1 -6343.693,E2 -6343.693} C_VEL
LIN {X 0,Y 495.726,Z 255.549,A -85,B 0,C 180,E1 -6346.302,E2 -6346.302} C_VEL
LIN {X 0,Y 495.772,Z 255.545,A -85,B 0,C 180,E1 -6349.3,E2 -6349.3} C_VEL
LIN {X 0,Y 495.754,Z 255.548,A -85,B 0,C 180,E1 -6351.408,E2 -6351.408} C_VEL
LIN {X 0,Y 495.747,Z 255.547,A -85,B 0,C 180,E1 -6354.461,E2 -6354.461} C_VEL
LIN {X 0,Y 495.757,Z 255.547,A -85,B 0,C 180,E1 -6357.404,E2 -6357.404} C_VEL
LIN {X 0,Y 495.751,Z 255.544,A -85,B 0,C 180,E1 -6360.741,E2 -6360.741} C_VEL
LIN {X 0,Y 495.089,Z 255.63,A -85,B 0,C 180,E1 -6361.42,E2 -6361.42} C_VEL
LIN {X 0,Y 492.232,Z 255.986,A -85,B 0,C 180,E1 -6362.523,E2 -6362.523} C_VEL
LIN {X 0,Y 489.824,Z 256.285,A -85,B 0,C 180,E1 -6363.412,E2 -6363.412} C_VEL
LIN {X 0,Y 488.806,Z 256.411,A -85,B 0,C 180,E1 -6364.098,E2 -6364.098} C_VEL
LIN {X 0,Y 488.732,Z 256.42,A -85,B 0,C 180,E1 -6364.33,E2 -6364.33} C_VEL
LIN {X 0,Y 488.733,Z 256.42,A -85,B 0,C 180,E1 -6367.153,E2 -6367.153} C_VEL
LIN {X 0,Y 488.708,Z 256.424,A -85,B 0,C 180,E1 -6369.809,E2 -6369.809} C_VEL
LIN {X 0,Y 488.544,Z 256.446,A -85,B 0,C 180,E1 -6372.415,E2 -6372.415} C_VEL
LIN {X 0,Y 488.321,Z 256.637,A -85,B 0,C 180,E1 -6374.129,E2 -6374.129} C_VEL
LIN {X 0,Y 488.323,Z 259.971,A -85,B 0,C 180,E1 -6376.686,E2 -6376.686} C_VEL
LIN {X 0,Y 488.375,Z 262.195,A -85,B 0,C 180,E1 -6378.376,E2 -6378.376} C_VEL
LIN {X 0,Y 488.247,Z 266.643,A -85,B 0,C 180,E1 -6381.723,E2 -6381.723} C_VEL
LIN {X 0,Y 488.194,Z 269.975,A -85,B 0,C 180,E1 -6384.215,E2 -6384.215} C_VEL
LIN {X 0,Y 488.183,Z 273.34,A -85,B 0,C 180,E1 -6386.698,E2 -6386.698} C_VEL
LIN {X 0,Y 487.95,Z 277.877,A -85,B 0,C 180,E1 -6389.999,E2 -6389.999} C_VEL
LIN {X 0,Y 487.977,Z 281.335,A -85,B 0,C 180,E1 -6392.501,E2 -6392.501} C_VEL
LIN {X 0,Y 489.726,Z 291.139,A -85,B 0,C 180,E1 -6392.878,E2 -6392.878} C_VEL
LIN {X 0,Y 489.585,Z 300.127,A -85,B 0,C 180,E1 -6393.291,E2 -6393.291} C_VEL
LIN {X 0,Y 489.356,Z 308.813,A -85,B 0,C 180,E1 -6393.807,E2 -6393.807} C_VEL
LIN {X 0,Y 489.075,Z 317.122,A -85,B 0,C 180,E1 -6394.429,E2 -6394.429} C_VEL
LIN {X 0,Y 488.843,Z 324.968,A -85,B 0,C 180,E1 -6395.154,E2 -6395.154} C_VEL
LIN {X 0,Y 488.654,Z 332.29,A -85,B 0,C 180,E1 -6395.984,E2 -6395.984} C_VEL
LIN {X 0,Y 488.508,Z 339.287,A -85,B 0,C 180,E1 -6396.959,E2 -6396.959} C_VEL
LIN {X 0,Y 488.289,Z 345.579,A -85,B 0,C 180,E1 -6398.066,E2 -6398.066} C_VEL
LIN {X 0,Y 488.12,Z 350.196,A -85,B 0,C 180,E1 -6399.112,E2 -6399.112} C_VEL
LIN {X 0,Y 488.042,Z 353.19,A -85,B 0,C 180,E1 -6399.95,E2 -6399.95} C_VEL
LIN {X 0,Y 487.994,Z 355.522,A -85,B 0,C 180,E1 -6400.79,E2 -6400.79} C_VEL
LIN {X 0,Y 487.975,Z 357.331,A -85,B 0,C 180,E1 -6401.674,E2 -6401.674} C_VEL
LIN {X 0,Y 487.91,Z 358.467,A -85,B 0,C 180,E1 -6402.477,E2 -6402.477} C_VEL
LIN {X 0,Y 487.871,Z 359.19,A -85,B 0,C 180,E1 -6403.325,E2 -6403.325} C_VEL
LIN {X 0,Y 487.881,Z 359.422,A -85,B 0,C 180,E1 -6404.174,E2 -6404.174} C_VEL
LIN {X 0,Y 487.893,Z 358.971,A -85,B 0,C 180,E1 -6405.187,E2 -6405.187} C_VEL
LIN {X 0,Y 487.935,Z 358.174,A -85,B 0,C 180,E1 -6405.881,E2 -6405.881} C_VEL
LIN {X 0,Y 487.999,Z 355.877,A -85,B 0,C 180,E1 -6407.17,E2 -6407.17} C_VEL
LIN {X 0,Y 488.129,Z 352.109,A -85,B 0,C 180,E1 -6408.465,E2 -6408.465} C_VEL
LIN {X 0,Y 488.223,Z 348.81,A -85,B 0,C 180,E1 -6409.333,E2 -6409.333} C_VEL
LIN {X 0,Y 488.367,Z 343.277,A -85,B 0,C 180,E1 -6410.463,E2 -6410.463} C_VEL
LIN {X 0,Y 488.517,Z 338.237,A -85,B 0,C 180,E1 -6411.299,E2 -6411.299} C_VEL
LIN {X 0,Y 488.728,Z 331.806,A -85,B 0,C 180,E1 -6412.176,E2 -6412.176} C_VEL
LIN {X 0,Y 488.909,Z 324.579,A -85,B 0,C 180,E1 -6412.987,E2 -6412.987} C_VEL
LIN {X 0,Y 489.175,Z 316.573,A -85,B 0,C 180,E1 -6413.719,E2 -6413.719} C_VEL
LIN {X 0,Y 489.511,Z 307.601,A -85,B 0,C 180,E1 -6414.378,E2 -6414.378} C_VEL
LIN {X 0,Y 489.718,Z 297.384,A -85,B 0,C 180,E1 -6414.954,E2 -6414.954} C_VEL
LIN {X 0,Y 489.559,Z 290.408,A -85,B 0,C 180,E1 -6415.262,E2 -6415.262} C_VEL
LIN {X 0,Y 487.975,Z 281.472,A -85,B 0,C 180,E1 -6415.598,E2 -6415.598} C_VEL
LIN {X 0,Y 487.987,Z 277.454,A -85,B 0,C 180,E1 -6418.541,E2 -6418.541} C_VEL
LIN {X 0,Y 488.051,Z 273.009,A -85,B 0,C 180,E1 -6421.836,E2 -6421.836} C_VEL
LIN {X 0,Y 488.065,Z 269.059,A -85,B 0,C 180,E1 -6424.841,E2 -6424.841} C_VEL
LIN {X 0,Y 488.164,Z 265.385,A -85,B 0,C 180,E1 -6427.648,E2 -6427.648} C_VEL
LIN {X 0,Y 488.25,Z 261.893,A -85,B 0,C 180,E1 -6430.37,E2 -6430.37} C_VEL
LIN {X 0,Y 488.366,Z 257.689,A -85,B 0,C 180,E1 -6433.688,E2 -6433.688} C_VEL
LIN {X 0,Y 488.41,Z 256.463,A -85,B 0,C 180,E1 -6434.835,E2 -6434.835} C_VEL
LIN {X 0,Y 488.653,Z 256.428,A -85,B 0,C 180,E1 -6437.473,E2 -6437.473} C_VEL
LIN {X 0,Y 488.715,Z 256.424,A -85,B 0,C 180,E1 -6439.678,E2 -6439.678} C_VEL
LIN {X 0,Y 488.665,Z 256.429,A -85,B 0,C 180,E1 -6442.278,E2 -6442.278} C_VEL
LIN {X 0,Y 488.709,Z 256.421,A -85,B 0,C 180,E1 -6445.052,E2 -6445.052} C_VEL
LIN {X 0,Y 488.684,Z 256.424,A -85,B 0,C 180,E1 -6448.047,E2 -6448.047} C_VEL
LIN {X 0,Y 488.705,Z 256.424,A -85,B 0,C 180,E1 -6450.731,E2 -6450.731} C_VEL
LIN {X 0,Y 488.739,Z 256.419,A -85,B 0,C 180,E1 -6453.529,E2 -6453.529} C_VEL
LIN {X 0,Y 488.67,Z 256.424,A -85,B 0,C 180,E1 -6456.256,E2 -6456.256} C_VEL
LIN {X 0,Y 488.729,Z 256.417,A -85,B 0,C 180,E1 -6459.177,E2 -6459.177} C_VEL
LIN {X 0,Y 488.743,Z 256.42,A -85,B 0,C 180,E1 -6461.629,E2 -6461.629} C_VEL
LIN {X 0,Y 488.745,Z 256.418,A -85,B 0,C 180,E1 -6465.001,E2 -6465.001} C_VEL
LIN {X 0,Y 488.817,Z 256.408,A -85,B 0,C 180,E1 -6468.39,E2 -6468.39} C_VEL
LIN {X 0,Y 488.803,Z 256.409,A -85,B 0,C 180,E1 -6471.735,E2 -6471.735} C_VEL
LIN {X 0,Y 488.796,Z 256.409,A -85,B 0,C 180,E1 -6475.053,E2 -6475.053} C_VEL
LIN {X 0,Y 488.952,Z 256.393,A -85,B 0,C 180,E1 -6477.53,E2 -6477.53} C_VEL
LIN {X 0,Y 488.955,Z 256.39,A -85,B 0,C 180,E1 -6480.001,E2 -6480.001} C_VEL
LIN {X 0,Y 488.948,Z 256.393,A -85,B 0,C 180,E1 -6482.473,E2 -6482.473} C_VEL
LIN {X 0,Y 488.846,Z 256.403,A -85,B 0,C 180,E1 -6485.777,E2 -6485.777} C_VEL
LIN {X 0,Y 488.805,Z 256.41,A -85,B 0,C 180,E1 -6488.268,E2 -6488.268} C_VEL
LIN {X 0,Y 488.819,Z 256.41,A -85,B 0,C 180,E1 -6491.613,E2 -6491.613} C_VEL
LIN {X 0,Y 488.753,Z 256.42,A -85,B 0,C 180,E1 -6495.002,E2 -6495.002} C_VEL
LIN {X 0,Y 488.736,Z 256.419,A -85,B 0,C 180,E1 -6498.444,E2 -6498.444} C_VEL
LIN {X 0,Y 488.7,Z 256.425,A -85,B 0,C 180,E1 -6501.072,E2 -6501.072} C_VEL
LIN {X 0,Y 488.685,Z 256.424,A -85,B 0,C 180,E1 -6503.747,E2 -6503.747} C_VEL
LIN {X 0,Y 488.713,Z 256.422,A -85,B 0,C 180,E1 -6506.476,E2 -6506.476} C_VEL
LIN {X 0,Y 488.703,Z 256.428,A -85,B 0,C 180,E1 -6509.273,E2 -6509.273} C_VEL
LIN {X 0,Y 488.699,Z 256.427,A -85,B 0,C 180,E1 -6512.148,E2 -6512.148} C_VEL
LIN {X 0,Y 488.709,Z 256.424,A -85,B 0,C 180,E1 -6515.117,E2 -6515.117} C_VEL
LIN {X 0,Y 488.674,Z 256.427,A -85,B 0,C 180,E1 -6518.201,E2 -6518.201} C_VEL
LIN {X 0,Y 488.745,Z 256.421,A -85,B 0,C 180,E1 -6520.35,E2 -6520.35} C_VEL
LIN {X 0,Y 488.679,Z 256.429,A -85,B 0,C 180,E1 -6523.656,E2 -6523.656} C_VEL
LIN {X 0,Y 488.68,Z 256.426,A -85,B 0,C 180,E1 -6526.347,E2 -6526.347} C_VEL
LIN {X 0,Y 488.729,Z 256.423,A -85,B 0,C 180,E1 -6529.678,E2 -6529.678} C_VEL
LIN {X 0,Y 488.675,Z 256.43,A -85,B 0,C 180,E1 -6532.842,E2 -6532.842} C_VEL
LIN {X 0,Y 488.711,Z 256.525,A -85,B 0,C 180,E1 -6534,E2 -6534} C_VEL
LIN {X 0,Y 489.662,Z 261.75,A -85,B 0,C 180,E1 -6536.353,E2 -6536.353} C_VEL
LIN {X 0,Y 489.796,Z 265.582,A -85,B 0,C 180,E1 -6537.935,E2 -6537.935} C_VEL
LIN {X 0,Y 489.401,Z 273.791,A -85,B 0,C 180,E1 -6541.163,E2 -6541.163} C_VEL
LIN {X 0,Y 488.965,Z 282.563,A -85,B 0,C 180,E1 -6544.458,E2 -6544.458} C_VEL
LIN {X 0,Y 488.674,Z 291.246,A -85,B 0,C 180,E1 -6547.598,E2 -6547.598} C_VEL
LIN {X 0,Y 488.384,Z 300.008,A -85,B 0,C 180,E1 -6550.673,E2 -6550.673} C_VEL
LIN {X 0,Y 488.282,Z 308.84,A -85,B 0,C 180,E1 -6553.701,E2 -6553.701} C_VEL
LIN {X 0,Y 488.112,Z 317.685,A -85,B 0,C 180,E1 -6556.682,E2 -6556.682} C_VEL
LIN {X 0,Y 488.114,Z 322.745,A -85,B 0,C 180,E1 -6558.372,E2 -6558.372} C_VEL
LIN {X 0,Y 489.441,Z 335.846,A -85,B 0,C 180,E1 -6558.824,E2 -6558.824} C_VEL
LIN {X 0,Y 489.378,Z 344.911,A -85,B 0,C 180,E1 -6559.241,E2 -6559.241} C_VEL
LIN {X 0,Y 489.171,Z 353.64,A -85,B 0,C 180,E1 -6559.76,E2 -6559.76} C_VEL
LIN {X 0,Y 488.928,Z 361.98,A -85,B 0,C 180,E1 -6560.382,E2 -6560.382} C_VEL
LIN {X 0,Y 488.676,Z 369.878,A -85,B 0,C 180,E1 -6561.107,E2 -6561.107} C_VEL
LIN {X 0,Y 488.419,Z 377.266,A -85,B 0,C 180,E1 -6561.936,E2 -6561.936} C_VEL
LIN {X 0,Y 488.218,Z 384.768,A -85,B 0,C 180,E1 -6562.973,E2 -6562.973} C_VEL
LIN {X 0,Y 488.121,Z 391.628,A -85,B 0,C 180,E1 -6564.217,E2 -6564.217} C_VEL
LIN {X 0,Y 487.951,Z 396.834,A -85,B 0,C 180,E1 -6565.458,E2 -6565.458} C_VEL
LIN {X 0,Y 487.985,Z 400.666,A -85,B 0,C 180,E1 -6566.699,E2 -6566.699} C_VEL
LIN {X 0,Y 487.936,Z 402.426,A -85,B 0,C 180,E1 -6567.525,E2 -6567.525} C_VEL
LIN {X 0,Y 487.892,Z 403.688,A -85,B 0,C 180,E1 -6568.35,E2 -6568.35} C_VEL
LIN {X 0,Y 487.834,Z 404.473,A -85,B 0,C 180,E1 -6569.176,E2 -6569.176} C_VEL
LIN {X 0,Y 487.824,Z 404.772,A -85,B 0,C 180,E1 -6570.001,E2 -6570.001} C_VEL
LIN {X 0,Y 487.834,Z 404.478,A -85,B 0,C 180,E1 -6570.827,E2 -6570.827} C_VEL
LIN {X 0,Y 487.892,Z 403.697,A -85,B 0,C 180,E1 -6571.652,E2 -6571.652} C_VEL
LIN {X 0,Y 487.936,Z 402.439,A -85,B 0,C 180,E1 -6572.478,E2 -6572.478} C_VEL
LIN {X 0,Y 488.006,Z 399.523,A -85,B 0,C 180,E1 -6573.717,E2 -6573.717} C_VEL
LIN {X 0,Y 487.951,Z 396.858,A -85,B 0,C 180,E1 -6574.545,E2 -6574.545} C_VEL
LIN {X 0,Y 488.122,Z 391.657,A -85,B 0,C 180,E1 -6575.785,E2 -6575.785} C_VEL
LIN {X 0,Y 488.28,Z 384.798,A -85,B 0,C 180,E1 -6577.028,E2 -6577.028} C_VEL
LIN {X 0,Y 488.424,Z 377.299,A -85,B 0,C 180,E1 -6578.066,E2 -6578.066} C_VEL
LIN {X 0,Y 488.678,Z 369.912,A -85,B 0,C 180,E1 -6578.895,E2 -6578.895} C_VEL
LIN {X 0,Y 488.923,Z 362.001,A -85,B 0,C 180,E1 -6579.62,E2 -6579.62} C_VEL
LIN {X 0,Y 489.131,Z 353.644,A -85,B 0,C 180,E1 -6580.243,E2 -6580.243} C_VEL
LIN {X 0,Y 489.471,Z 342.977,A -85,B 0,C 180,E1 -6580.864,E2 -6580.864} C_VEL
LIN {X 0,Y 489.408,Z 335.794,A -85,B 0,C 180,E1 -6581.179,E2 -6581.179} C_VEL
LIN {X 0,Y 488.105,Z 322.834,A -85,B 0,C 180,E1 -6581.63,E2 -6581.63} C_VEL
LIN {X 0,Y 488.215,Z 312.682,A -85,B 0,C 180,E1 -6585.019,E2 -6585.019} C_VEL
LIN {X 0,Y 488.368,Z 303.201,A -85,B 0,C 180,E1 -6588.232,E2 -6588.232} C_VEL
LIN {X 0,Y 488.573,Z 293.662,A -85,B 0,C 180,E1 -6591.52,E2 -6591.52} C_VEL
LIN {X 0,Y 488.796,Z 286.066,A -85,B 0,C 180,E1 -6594.192,E2 -6594.192} C_VEL
LIN {X 0,Y 489.13,Z 277.23,A -85,B 0,C 180,E1 -6597.374,E2 -6597.374} C_VEL
LIN {X 0,Y 489.453,Z 268.78,A -85,B 0,C 180,E1 -6600.51,E2 -6600.51} C_VEL
LIN {X 0,Y 489.632,Z 262.166,A -85,B 0,C 180,E1 -6603.056,E2 -6603.056} C_VEL
LIN {X 0,Y 488.759,Z 256.419,A -85,B 0,C 180,E1 -6605.491,E2 -6605.491} C_VEL
LIN {X 0,Y 488.711,Z 256.424,A -85,B 0,C 180,E1 -6609.053,E2 -6609.053} C_VEL
LIN {X 0,Y 488.715,Z 256.424,A -85,B 0,C 180,E1 -6611.6,E2 -6611.6} C_VEL
LIN {X 0,Y 488.709,Z 256.422,A -85,B 0,C 180,E1 -6614.803,E2 -6614.803} C_VEL
LIN {X 0,Y 488.7,Z 256.426,A -85,B 0,C 180,E1 -6617.474,E2 -6617.474} C_VEL
LIN {X 0,Y 488.742,Z 256.421,A -85,B 0,C 180,E1 -6619.677,E2 -6619.677} C_VEL
LIN {X 0,Y 488.678,Z 256.427,A -85,B 0,C 180,E1 -6622.84,E2 -6622.84} C_VEL
LIN {X 0,Y 488.738,Z 256.42,A -85,B 0,C 180,E1 -6625.887,E2 -6625.887} C_VEL
LIN {X 0,Y 488.701,Z 256.425,A -85,B 0,C 180,E1 -6628.82,E2 -6628.82} C_VEL
LIN {X 0,Y 488.752,Z 256.419,A -85,B 0,C 180,E1 -6631.671,E2 -6631.671} C_VEL
LIN {X 0,Y 488.736,Z 256.42,A -85,B 0,C 180,E1 -6634.443,E2 -6634.443} C_VEL
LIN {X 0,Y 488.73,Z 256.421,A -85,B 0,C 180,E1 -6637.152,E2 -6637.152} C_VEL
LIN {X 0,Y 488.733,Z 256.42,A -85,B 0,C 180,E1 -6639.81,E2 -6639.81} C_VEL
LIN {X 0,Y 488.722,Z 256.421,A -85,B 0,C 180,E1 -6642.422,E2 -6642.422} C_VEL
LIN {X 0,Y 488.769,Z 256.417,A -85,B 0,C 180,E1 -6644.999,E2 -6644.999} C_VEL
LIN {X 0,Y 488.813,Z 256.41,A -85,B 0,C 180,E1 -6648.386,E2 -6648.386} C_VEL
LIN {X 0,Y 488.792,Z 256.413,A -85,B 0,C 180,E1 -6651.732,E2 -6651.732} C_VEL
LIN {X 0,Y 488.852,Z 256.406,A -85,B 0,C 180,E1 -6654.223,E2 -6654.223} C_VEL
LIN {X 0,Y 488.966,Z 256.391,A -85,B 0,C 180,E1 -6657.527,E2 -6657.527} C_VEL
LIN {X 0,Y 488.96,Z 256.394,A -85,B 0,C 180,E1 -6660.822,E2 -6660.822} C_VEL
LIN {X 0,Y 488.966,Z 256.392,A -85,B 0,C 180,E1 -6662.47,E2 -6662.47} C_VEL
LIN {X 0,Y 488.859,Z 256.404,A -85,B 0,C 180,E1 -6665.774,E2 -6665.774} C_VEL
LIN {X 0,Y 488.821,Z 256.411,A -85,B 0,C 180,E1 -6668.265,E2 -6668.265} C_VEL
LIN {X 0,Y 488.808,Z 256.41,A -85,B 0,C 180,E1 -6671.611,E2 -6671.611} C_VEL
LIN {X 0,Y 488.764,Z 256.417,A -85,B 0,C 180,E1 -6674.998,E2 -6674.998} C_VEL
LIN {X 0,Y 488.756,Z 256.418,A -85,B 0,C 180,E1 -6678.44,E2 -6678.44} C_VEL
LIN {X 0,Y 488.707,Z 256.423,A -85,B 0,C 180,E1 -6681.069,E2 -6681.069} C_VEL
LIN {X 0,Y 488.692,Z 256.426,A -85,B 0,C 180,E1 -6683.743,E2 -6683.743} C_VEL
LIN {X 0,Y 488.79,Z 256.412,A -85,B 0,C 180,E1 -6686.942,E2 -6686.942} C_VEL
LIN {X 0,Y 488.707,Z 256.423,A -85,B 0,C 180,E1 -6690.361,E2 -6690.361} C_VEL
LIN {X 0,Y 488.732,Z 256.422,A -85,B 0,C 180,E1 -6693.482,E2 -6693.482} C_VEL
LIN {X 0,Y 488.683,Z 256.427,A -85,B 0,C 180,E1 -6696.354,E2 -6696.354} C_VEL
LIN {X 0,Y 488.736,Z 256.421,A -85,B 0,C 180,E1 -6699.248,E2 -6699.248} C_VEL
LIN {X 0,Y 488.727,Z 256.421,A -85,B 0,C 180,E1 -6702.519,E2 -6702.519} C_VEL
LIN {X 0,Y 488.693,Z 256.425,A -85,B 0,C 180,E1 -6705.974,E2 -6705.974} C_VEL
LIN {X 0,Y 488.717,Z 256.423,A -85,B 0,C 180,E1 -6708.584,E2 -6708.584} C_VEL
LIN {X 0,Y 488.737,Z 256.421,A -85,B 0,C 180,E1 -6710.939,E2 -6710.939} C_VEL
LIN {X 0,Y 488.675,Z 256.426,A -85,B 0,C 180,E1 -6713.867,E2 -6713.867} C_VEL
LIN {X 0,Y 488.727,Z 256.422,A -85,B 0,C 180,E1 -6716.875,E2 -6716.875} C_VEL
LIN {X 0,Y 488.72,Z 256.422,A -85,B 0,C 180,E1 -6719.78,E2 -6719.78} C_VEL
LIN {X 0,Y 488.784,Z 256.414,A -85,B 0,C 180,E1 -6723.053,E2 -6723.053} C_VEL
LIN {X 0,Y 488.732,Z 256.42,A -85,B 0,C 180,E1 -6724.33,E2 -6724.33} C_VEL
LIN {X 0,Y 488.085,Z 256.504,A -85,B 0,C 180,E1 -6725.018,E2 -6725.018} C_VEL
LIN {X 0,Y 485.224,Z 256.861,A -85,B 0,C 180,E1 -6726.135,E2 -6726.135} C_VEL
LIN {X 0,Y 482.787,Z 257.162,A -85,B 0,C 180,E1 -6727.034,E2 -6727.034} C_VEL
LIN {X 0,Y 481.735,Z 257.292,A -85,B 0,C 180,E1 -6727.73,E2 -6727.73} C_VEL
LIN {X 0,Y 481.647,Z 257.302,A -85,B 0,C 180,E1 -6727.965,E2 -6727.965} C_VEL
LIN {X 0,Y 481.673,Z 257.301,A -85,B 0,C 180,E1 -6730.391,E2 -6730.391} C_VEL
LIN {X 0,Y 481.543,Z 257.318,A -85,B 0,C 180,E1 -6732.151,E2 -6732.151} C_VEL
LIN {X 0,Y 481.286,Z 257.35,A -85,B 0,C 180,E1 -6733.891,E2 -6733.891} C_VEL
LIN {X 0,Y 481.314,Z 258.154,A -85,B 0,C 180,E1 -6734.761,E2 -6734.761} C_VEL
LIN {X 0,Y 481.34,Z 262.616,A -85,B 0,C 180,E1 -6738.204,E2 -6738.204} C_VEL
LIN {X 0,Y 481.175,Z 267.09,A -85,B 0,C 180,E1 -6741.6,E2 -6741.6} C_VEL
LIN {X 0,Y 481.14,Z 270.475,A -85,B 0,C 180,E1 -6744.13,E2 -6744.13} C_VEL
LIN {X 0,Y 481.131,Z 273.854,A -85,B 0,C 180,E1 -6746.649,E2 -6746.649} C_VEL
LIN {X 0,Y 480.871,Z 278.427,A -85,B 0,C 180,E1 -6749.999,E2 -6749.999} C_VEL
LIN {X 0,Y 480.893,Z 281.634,A -85,B 0,C 180,E1 -6752.328,E2 -6752.328} C_VEL
LIN {X 0,Y 482.773,Z 292.371,A -85,B 0,C 180,E1 -6752.763,E2 -6752.763} C_VEL
LIN {X 0,Y 482.61,Z 300.248,A -85,B 0,C 180,E1 -6753.129,E2 -6753.129} C_VEL
LIN {X 0,Y 482.399,Z 308.966,A -85,B 0,C 180,E1 -6753.653,E2 -6753.653} C_VEL
LIN {X 0,Y 482.086,Z 317.314,A -85,B 0,C 180,E1 -6754.284,E2 -6754.284} C_VEL
LIN {X 0,Y 481.854,Z 325.179,A -85,B 0,C 180,E1 -6755.019,E2 -6755.019} C_VEL
LIN {X 0,Y 481.63,Z 332.529,A -85,B 0,C 180,E1 -6755.862,E2 -6755.862} C_VEL
LIN {X 0,Y 481.441,Z 340.336,A -85,B 0,C 180,E1 -6756.972,E2 -6756.972} C_VEL
LIN {X 0,Y 481.247,Z 345.858,A -85,B 0,C 180,E1 -6757.973,E2 -6757.973} C_VEL
LIN {X 0,Y 481.077,Z 349.691,A -85,B 0,C 180,E1 -6758.822,E2 -6758.822} C_VEL
LIN {X 0,Y 480.965,Z 354.078,A -85,B 0,C 180,E1 -6760.098,E2 -6760.098} C_VEL
LIN {X 0,Y 480.901,Z 356.328,A -85,B 0,C 180,E1 -6760.951,E2 -6760.951} C_VEL
LIN {X 0,Y 480.871,Z 357.97,A -85,B 0,C 180,E1 -6761.806,E2 -6761.806} C_VEL
LIN {X 0,Y 480.808,Z 359.033,A -85,B 0,C 180,E1 -6762.664,E2 -6762.664} C_VEL
LIN {X 0,Y 480.773,Z 359.599,A -85,B 0,C 180,E1 -6763.525,E2 -6763.525} C_VEL
LIN {X 0,Y 480.812,Z 359.673,A -85,B 0,C 180,E1 -6764.387,E2 -6764.387} C_VEL
LIN {X 0,Y 480.807,Z 359.231,A -85,B 0,C 180,E1 -6765.273,E2 -6765.273} C_VEL
LIN {X 0,Y 480.858,Z 358.263,A -85,B 0,C 180,E1 -6766.121,E2 -6766.121} C_VEL
LIN {X 0,Y 480.927,Z 355.675,A -85,B 0,C 180,E1 -6767.431,E2 -6767.431} C_VEL
LIN {X 0,Y 481.022,Z 353.394,A -85,B 0,C 180,E1 -6768.261,E2 -6768.261} C_VEL
LIN {X 0,Y 481.159,Z 350.107,A -85,B 0,C 180,E1 -6769.185,E2 -6769.185} C_VEL
LIN {X 0,Y 481.302,Z 345.118,A -85,B 0,C 180,E1 -6770.29,E2 -6770.29} C_VEL
LIN {X 0,Y 481.488,Z 338.643,A -85,B 0,C 180,E1 -6771.401,E2 -6771.401} C_VEL
LIN {X 0,Y 481.704,Z 332.23,A -85,B 0,C 180,E1 -6772.291,E2 -6772.291} C_VEL
LIN {X 0,Y 481.916,Z 325.41,A -85,B 0,C 180,E1 -6773.073,E2 -6773.073} C_VEL
LIN {X 0,Y 482.175,Z 318.368,A -85,B 0,C 180,E1 -6773.742,E2 -6773.742} C_VEL
LIN {X 0,Y 482.413,Z 311.291,A -85,B 0,C 180,E1 -6774.301,E2 -6774.301} C_VEL
LIN {X 0,Y 482.649,Z 302.506,A -85,B 0,C 180,E1 -6774.862,E2 -6774.862} C_VEL
LIN {X 0,Y 482.841,Z 293.088,A -85,B 0,C 180,E1 -6775.325,E2 -6775.325} C_VEL
LIN {X 0,Y 481.111,Z 283.165,A -85,B 0,C 180,E1 -6775.73,E2 -6775.73} C_VEL
LIN {X 0,Y 480.896,Z 281.761,A -85,B 0,C 180,E1 -6775.806,E2 -6775.806} C_VEL
LIN {X 0,Y 480.908,Z 277.67,A -85,B 0,C 180,E1 -6778.832,E2 -6778.832} C_VEL
LIN {X 0,Y 480.997,Z 273.351,A -85,B 0,C 180,E1 -6782.069,E2 -6782.069} C_VEL
LIN {X 0,Y 481.042,Z 269.382,A -85,B 0,C 180,E1 -6785.104,E2 -6785.104} C_VEL
LIN {X 0,Y 481.095,Z 265.768,A -85,B 0,C 180,E1 -6787.926,E2 -6787.926} C_VEL
LIN {X 0,Y 481.221,Z 261.754,A -85,B 0,C 180,E1 -6791.085,E2 -6791.085} C_VEL
LIN {X 0,Y 481.336,Z 257.513,A -85,B 0,C 180,E1 -6794.493,E2 -6794.493} C_VEL
LIN {X 0,Y 481.57,Z 257.31,A -85,B 0,C 180,E1 -6796.859,E2 -6796.859} C_VEL
LIN {X 0,Y 481.672,Z 257.298,A -85,B 0,C 180,E1 -6800.062,E2 -6800.062} C_VEL
LIN {X 0,Y 481.612,Z 257.306,A -85,B 0,C 180,E1 -6803.255,E2 -6803.255} C_VEL
LIN {X 0,Y 481.69,Z 257.296,A -85,B 0,C 180,E1 -6806.331,E2 -6806.331} C_VEL
LIN {X 0,Y 481.631,Z 257.304,A -85,B 0,C 180,E1 -6809.418,E2 -6809.418} C_VEL
LIN {X 0,Y 481.682,Z 257.301,A -85,B 0,C 180,E1 -6812.169,E2 -6812.169} C_VEL
LIN {X 0,Y 481.694,Z 257.296,A -85,B 0,C 180,E1 -6814.971,E2 -6814.971} C_VEL
LIN {X 0,Y 481.632,Z 257.302,A -85,B 0,C 180,E1 -6817.706,E2 -6817.706} C_VEL
LIN {X 0,Y 481.692,Z 257.297,A -85,B 0,C 180,E1 -6820.395,E2 -6820.395} C_VEL
LIN {X 0,Y 481.675,Z 257.297,A -85,B 0,C 180,E1 -6823.035,E2 -6823.035} C_VEL
LIN {X 0,Y 481.673,Z 257.295,A -85,B 0,C 180,E1 -6825.64,E2 -6825.64} C_VEL
LIN {X 0,Y 481.781,Z 257.286,A -85,B 0,C 180,E1 -6828.218,E2 -6828.218} C_VEL
LIN {X 0,Y 481.749,Z 257.289,A -85,B 0,C 180,E1 -6831.613,E2 -6831.613} C_VEL
LIN {X 0,Y 481.765,Z 257.285,A -85,B 0,C 180,E1 -6834.98,E2 -6834.98} C_VEL
LIN {X 0,Y 481.918,Z 257.269,A -85,B 0,C 180,E1 -6837.494,E2 -6837.494} C_VEL
LIN {X 0,Y 481.927,Z 257.265,A -85,B 0,C 180,E1 -6840.002,E2 -6840.002} C_VEL
LIN {X 0,Y 481.915,Z 257.269,A -85,B 0,C 180,E1 -6842.509,E2 -6842.509} C_VEL
LIN {X 0,Y 481.807,Z 257.279,A -85,B 0,C 180,E1 -6845.862,E2 -6845.862} C_VEL
LIN {X 0,Y 481.751,Z 257.29,A -85,B 0,C 180,E1 -6848.39,E2 -6848.39} C_VEL
LIN {X 0,Y 481.785,Z 257.288,A -85,B 0,C 180,E1 -6851.785,E2 -6851.785} C_VEL
LIN {X 0,Y 481.734,Z 257.292,A -85,B 0,C 180,E1 -6855.226,E2 -6855.226} C_VEL
LIN {X 0,Y 481.698,Z 257.294,A -85,B 0,C 180,E1 -6858.723,E2 -6858.723} C_VEL
LIN {X 0,Y 481.64,Z 257.305,A -85,B 0,C 180,E1 -6861.396,E2 -6861.396} C_VEL
LIN {X 0,Y 481.667,Z 257.3,A -85,B 0,C 180,E1 -6864.115,E2 -6864.115} C_VEL
LIN {X 0,Y 481.687,Z 257.297,A -85,B 0,C 180,E1 -6867.128,E2 -6867.128} C_VEL
LIN {X 0,Y 481.666,Z 257.3,A -85,B 0,C 180,E1 -6869.743,E2 -6869.743} C_VEL
LIN {X 0,Y 481.667,Z 257.303,A -85,B 0,C 180,E1 -6872.676,E2 -6872.676} C_VEL
LIN {X 0,Y 481.625,Z 257.308,A -85,B 0,C 180,E1 -6875.711,E2 -6875.711} C_VEL
LIN {X 0,Y 481.709,Z 257.294,A -85,B 0,C 180,E1 -6879.355,E2 -6879.355} C_VEL
LIN {X 0,Y 481.644,Z 257.304,A -85,B 0,C 180,E1 -6882.162,E2 -6882.162} C_VEL
LIN {X 0,Y 481.65,Z 257.302,A -85,B 0,C 180,E1 -6885.544,E2 -6885.544} C_VEL
LIN {X 0,Y 481.653,Z 257.302,A -85,B 0,C 180,E1 -6888.96,E2 -6888.96} C_VEL
LIN {X 0,Y 481.65,Z 257.304,A -85,B 0,C 180,E1 -6891.994,E2 -6891.994} C_VEL
LIN {X 0,Y 481.651,Z 257.456,A -85,B 0,C 180,E1 -6893.777,E2 -6893.777} C_VEL
LIN {X 0,Y 482.712,Z 263.226,A -85,B 0,C 180,E1 -6896.411,E2 -6896.411} C_VEL
LIN {X 0,Y 482.752,Z 267.97,A -85,B 0,C 180,E1 -6898.394,E2 -6898.394} C_VEL
LIN {X 0,Y 482.282,Z 276.383,A -85,B 0,C 180,E1 -6901.733,E2 -6901.733} C_VEL
LIN {X 0,Y 481.869,Z 284.943,A -85,B 0,C 180,E1 -6904.98,E2 -6904.98} C_VEL
LIN {X 0,Y 481.596,Z 292.341,A -85,B 0,C 180,E1 -6907.704,E2 -6907.704} C_VEL
LIN {X 0,Y 481.32,Z 301.086,A -85,B 0,C 180,E1 -6910.822,E2 -6910.822} C_VEL
LIN {X 0,Y 481.215,Z 309.872,A -85,B 0,C 180,E1 -6913.891,E2 -6913.891} C_VEL
LIN {X 0,Y 481.007,Z 318.664,A -85,B 0,C 180,E1 -6916.912,E2 -6916.912} C_VEL
LIN {X 0,Y 481.026,Z 322.538,A -85,B 0,C 180,E1 -6918.21,E2 -6918.21} C_VEL
LIN {X 0,Y 482.282,Z 334.773,A -85,B 0,C 180,E1 -6918.617,E2 -6918.617} C_VEL
LIN {X 0,Y 482.497,Z 342.842,A -85,B 0,C 180,E1 -6918.983,E2 -6918.983} C_VEL
LIN {X 0,Y 482.189,Z 353.381,A -85,B 0,C 180,E1 -6919.61,E2 -6919.61} C_VEL
LIN {X 0,Y 481.9,Z 361.7,A -85,B 0,C 180,E1 -6920.24,E2 -6920.24} C_VEL
LIN {X 0,Y 481.635,Z 369.582,A -85,B 0,C 180,E1 -6920.976,E2 -6920.976} C_VEL
LIN {X 0,Y 481.381,Z 376.96,A -85,B 0,C 180,E1 -6921.818,E2 -6921.818} C_VEL
LIN {X 0,Y 481.158,Z 384.453,A -85,B 0,C 180,E1 -6922.869,E2 -6922.869} C_VEL
LIN {X 0,Y 481.021,Z 391.303,A -85,B 0,C 180,E1 -6924.131,E2 -6924.131} C_VEL
LIN {X 0,Y 480.868,Z 396.508,A -85,B 0,C 180,E1 -6925.391,E2 -6925.391} C_VEL
LIN {X 0,Y 480.914,Z 400.339,A -85,B 0,C 180,E1 -6926.65,E2 -6926.65} C_VEL
LIN {X 0,Y 480.849,Z 402.098,A -85,B 0,C 180,E1 -6927.488,E2 -6927.488} C_VEL
LIN {X 0,Y 480.823,Z 403.36,A -85,B 0,C 180,E1 -6928.326,E2 -6928.326} C_VEL
LIN {X 0,Y 480.76,Z 404.144,A -85,B 0,C 180,E1 -6929.163,E2 -6929.163} C_VEL
LIN {X 0,Y 480.747,Z 404.444,A -85,B 0,C 180,E1 -6930.001,E2 -6930.001} C_VEL
LIN {X 0,Y 480.76,Z 404.15,A -85,B 0,C 180,E1 -6930.839,E2 -6930.839} C_VEL
LIN {X 0,Y 480.823,Z 403.367,A -85,B 0,C 180,E1 -6931.676,E2 -6931.676} C_VEL
LIN {X 0,Y 480.849,Z 402.107,A -85,B 0,C 180,E1 -6932.514,E2 -6932.514} C_VEL
LIN {X 0,Y 480.925,Z 399.19,A -85,B 0,C 180,E1 -6933.772,E2 -6933.772} C_VEL
LIN {X 0,Y 480.869,Z 396.523,A -85,B 0,C 180,E1 -6934.612,E2 -6934.612} C_VEL
LIN {X 0,Y 481.022,Z 391.317,A -85,B 0,C 180,E1 -6935.871,E2 -6935.871} C_VEL
LIN {X 0,Y 481.209,Z 384.452,A -85,B 0,C 180,E1 -6937.132,E2 -6937.132} C_VEL
LIN {X 0,Y 481.385,Z 376.946,A -85,B 0,C 180,E1 -6938.185,E2 -6938.185} C_VEL
LIN {X 0,Y 481.618,Z 369.546,A -85,B 0,C 180,E1 -6939.026,E2 -6939.026} C_VEL
LIN {X 0,Y 481.885,Z 361.623,A -85,B 0,C 180,E1 -6939.762,E2 -6939.762} C_VEL
LIN {X 0,Y 482.142,Z 353.25,A -85,B 0,C 180,E1 -6940.393,E2 -6940.393} C_VEL
LIN {X 0,Y 482.489,Z 342.678,A -85,B 0,C 180,E1 -6941.016,E2 -6941.016} C_VEL
LIN {X 0,Y 482.349,Z 335.936,A -85,B 0,C 180,E1 -6941.319,E2 -6941.319} C_VEL
LIN {X 0,Y 481.002,Z 322.595,A -85,B 0,C 180,E1 -6941.776,E2 -6941.776} C_VEL
LIN {X 0,Y 481.133,Z 312.385,A -85,B 0,C 180,E1 -6945.245,E2 -6945.245} C_VEL
LIN {X 0,Y 481.287,Z 303.395,A -85,B 0,C 180,E1 -6948.347,E2 -6948.347} C_VEL
LIN {X 0,Y 481.491,Z 294.666,A -85,B 0,C 180,E1 -6951.403,E2 -6951.403} C_VEL
LIN {X 0,Y 481.74,Z 287.086,A -85,B 0,C 180,E1 -6954.111,E2 -6954.111} C_VEL
LIN {X 0,Y 482.067,Z 278.593,A -85,B 0,C 180,E1 -6957.212,E2 -6957.212} C_VEL
LIN {X 0,Y 482.403,Z 270.726,A -85,B 0,C 180,E1 -6960.175,E2 -6960.175} C_VEL
LIN {X 0,Y 482.653,Z 264.468,A -85,B 0,C 180,E1 -6962.6,E2 -6962.6} C_VEL
LIN {X 0,Y 482.415,Z 261.36,A -85,B 0,C 180,E1 -6963.86,E2 -6963.86} C_VEL
LIN {X 0,Y 481.697,Z 257.299,A -85,B 0,C 180,E1 -6965.636,E2 -6965.636} C_VEL
LIN {X 0,Y 481.678,Z 257.299,A -85,B 0,C 180,E1 -6968.859,E2 -6968.859} C_VEL
LIN {X 0,Y 481.66,Z 257.302,A -85,B 0,C 180,E1 -6971.913,E2 -6971.913} C_VEL
LIN {X 0,Y 481.663,Z 257.301,A -85,B 0,C 180,E1 -6974.458,E2 -6974.458} C_VEL
LIN {X 0,Y 481.656,Z 257.303,A -85,B 0,C 180,E1 -6977.839,E2 -6977.839} C_VEL
LIN {X 0,Y 481.669,Z 257.3,A -85,B 0,C 180,E1 -6980.654,E2 -6980.654} C_VEL
LIN {X 0,Y 481.63,Z 257.306,A -85,B 0,C 180,E1 -6983.377,E2 -6983.377} C_VEL
LIN {X 0,Y 481.702,Z 257.297,A -85,B 0,C 180,E1 -6986.328,E2 -6986.328} C_VEL
LIN {X 0,Y 481.659,Z 257.303,A -85,B 0,C 180,E1 -6989.417,E2 -6989.417} C_VEL
LIN {X 0,Y 481.708,Z 257.295,A -85,B 0,C 180,E1 -6992.167,E2 -6992.167} C_VEL
LIN {X 0,Y 481.702,Z 257.297,A -85,B 0,C 180,E1 -6994.968,E2 -6994.968} C_VEL
LIN {X 0,Y 481.657,Z 257.302,A -85,B 0,C 180,E1 -6997.704,E2 -6997.704} C_VEL
LIN {X 0,Y 481.713,Z 257.293,A -85,B 0,C 180,E1 -7000.392,E2 -7000.392} C_VEL
LIN {X 0,Y 481.686,Z 257.299,A -85,B 0,C 180,E1 -7003.033,E2 -7003.033} C_VEL
LIN {X 0,Y 481.696,Z 257.298,A -85,B 0,C 180,E1 -7005.638,E2 -7005.638} C_VEL
LIN {X 0,Y 481.758,Z 257.289,A -85,B 0,C 180,E1 -7008.214,E2 -7008.214} C_VEL
LIN {X 0,Y 481.746,Z 257.291,A -85,B 0,C 180,E1 -7011.61,E2 -7011.61} C_VEL
LIN {X 0,Y 481.813,Z 257.283,A -85,B 0,C 180,E1 -7014.138,E2 -7014.138} C_VEL
LIN {X 0,Y 481.933,Z 257.267,A -85,B 0,C 180,E1 -7017.491,E2 -7017.491} C_VEL
LIN {X 0,Y 481.911,Z 257.272,A -85,B 0,C 180,E1 -7020.834,E2 -7020.834} C_VEL
LIN {X 0,Y 481.933,Z 257.268,A -85,B 0,C 180,E1 -7022.506,E2 -7022.506} C_VEL
LIN {X 0,Y 481.82,Z 257.281,A -85,B 0,C 180,E1 -7025.859,E2 -7025.859} C_VEL
LIN {X 0,Y 481.767,Z 257.289,A -85,B 0,C 180,E1 -7028.387,E2 -7028.387} C_VEL
LIN {X 0,Y 481.754,Z 257.29,A -85,B 0,C 180,E1 -7031.783,E2 -7031.783} C_VEL
LIN {X 0,Y 481.744,Z 257.291,A -85,B 0,C 180,E1 -7035.222,E2 -7035.222} C_VEL
LIN {X 0,Y 481.713,Z 257.295,A -85,B 0,C 180,E1 -7038.72,E2 -7038.72} C_VEL
LIN {X 0,Y 481.646,Z 257.304,A -85,B 0,C 180,E1 -7041.393,E2 -7041.393} C_VEL
LIN {X 0,Y 481.676,Z 257.302,A -85,B 0,C 180,E1 -7044.111,E2 -7044.111} C_VEL
LIN {X 0,Y 481.745,Z 257.29,A -85,B 0,C 180,E1 -7047.137,E2 -7047.137} C_VEL
LIN {X 0,Y 481.676,Z 257.3,A -85,B 0,C 180,E1 -7049.739,E2 -7049.739} C_VEL
LIN {X 0,Y 481.669,Z 257.299,A -85,B 0,C 180,E1 -7052.672,E2 -7052.672} C_VEL
LIN {X 0,Y 481.638,Z 257.305,A -85,B 0,C 180,E1 -7055.707,E2 -7055.707} C_VEL
LIN {X 0,Y 481.707,Z 257.297,A -85,B 0,C 180,E1 -7059.352,E2 -7059.352} C_VEL
LIN {X 0,Y 481.667,Z 257.301,A -85,B 0,C 180,E1 -7062.156,E2 -7062.156} C_VEL
LIN {X 0,Y 481.651,Z 257.302,A -85,B 0,C 180,E1 -7064.455,E2 -7064.455} C_VEL
LIN {X 0,Y 481.68,Z 257.3,A -85,B 0,C 180,E1 -7066.844,E2 -7066.844} C_VEL
LIN {X 0,Y 481.683,Z 257.297,A -85,B 0,C 180,E1 -7070.059,E2 -7070.059} C_VEL
LIN {X 0,Y 481.62,Z 257.308,A -85,B 0,C 180,E1 -7073.252,E2 -7073.252} C_VEL
LIN {X 0,Y 481.697,Z 257.296,A -85,B 0,C 180,E1 -7076.328,E2 -7076.328} C_VEL
LIN {X 0,Y 481.645,Z 257.304,A -85,B 0,C 180,E1 -7079.414,E2 -7079.414} C_VEL
LIN {X 0,Y 481.688,Z 257.298,A -85,B 0,C 180,E1 -7082.166,E2 -7082.166} C_VEL
LIN {X 0,Y 481.704,Z 257.296,A -85,B 0,C 180,E1 -7084.968,E2 -7084.968} C_VEL
LIN {X 0,Y 481.647,Z 257.302,A -85,B 0,C 180,E1 -7087.965,E2 -7087.965} C_VEL
LIN {X 0,Y 480.985,Z 257.388,A -85,B 0,C 180,E1 -7088.663,E2 -7088.663} C_VEL
LIN {X 0,Y 478.158,Z 257.738,A -85,B 0,C 180,E1 -7089.797,E2 -7089.797} C_VEL
LIN {X 0,Y 475.744,Z 258.04,A -85,B 0,C 180,E1 -7090.71,E2 -7090.71} C_VEL
LIN {X 0,Y 474.672,Z 258.171,A -85,B 0,C 180,E1 -7091.416,E2 -7091.416} C_VEL
LIN {X 0,Y 474.566,Z 258.184,A -85,B 0,C 180,E1 -7091.655,E2 -7091.655} C_VEL
LIN {X 0,Y 474.247,Z 258.396,A -85,B 0,C 180,E1 -7094.409,E2 -7094.409} C_VEL
LIN {X 0,Y 474.274,Z 263.055,A -85,B 0,C 180,E1 -7098.026,E2 -7098.026} C_VEL
LIN {X 0,Y 474.118,Z 267.559,A -85,B 0,C 180,E1 -7101.474,E2 -7101.474} C_VEL
LIN {X 0,Y 474.086,Z 270.955,A -85,B 0,C 180,E1 -7104.043,E2 -7104.043} C_VEL
LIN {X 0,Y 474.08,Z 274.368,A -85,B 0,C 180,E1 -7106.599,E2 -7106.599} C_VEL
LIN {X 0,Y 473.792,Z 278.978,A -85,B 0,C 180,E1 -7109.999,E2 -7109.999} C_VEL
LIN {X 0,Y 473.811,Z 281.956,A -85,B 0,C 180,E1 -7112.177,E2 -7112.177} C_VEL
LIN {X 0,Y 475.67,Z 292.396,A -85,B 0,C 180,E1 -7112.592,E2 -7112.592} C_VEL
LIN {X 0,Y 475.594,Z 302.126,A -85,B 0,C 180,E1 -7113.07,E2 -7113.07} C_VEL
LIN {X 0,Y 475.33,Z 310.557,A -85,B 0,C 180,E1 -7113.602,E2 -7113.602} C_VEL
LIN {X 0,Y 475.039,Z 318.671,A -85,B 0,C 180,E1 -7114.241,E2 -7114.241} C_VEL
LIN {X 0,Y 474.812,Z 326.363,A -85,B 0,C 180,E1 -7114.988,E2 -7114.988} C_VEL
LIN {X 0,Y 474.572,Z 334.421,A -85,B 0,C 180,E1 -7115.949,E2 -7115.949} C_VEL
LIN {X 0,Y 474.387,Z 341.361,A -85,B 0,C 180,E1 -7116.998,E2 -7116.998} C_VEL
LIN {X 0,Y 474.145,Z 347.082,A -85,B 0,C 180,E1 -7118.094,E2 -7118.094} C_VEL
LIN {X 0,Y 473.952,Z 352.292,A -85,B 0,C 180,E1 -7119.386,E2 -7119.386} C_VEL
LIN {X 0,Y 473.855,Z 356.113,A -85,B 0,C 180,E1 -7120.683,E2 -7120.683} C_VEL
LIN {X 0,Y 473.773,Z 358.605,A -85,B 0,C 180,E1 -7121.985,E2 -7121.985} C_VEL
LIN {X 0,Y 473.704,Z 359.593,A -85,B 0,C 180,E1 -7122.857,E2 -7122.857} C_VEL
LIN {X 0,Y 473.684,Z 360.007,A -85,B 0,C 180,E1 -7123.731,E2 -7123.731} C_VEL
LIN {X 0,Y 473.709,Z 359.928,A -85,B 0,C 180,E1 -7124.607,E2 -7124.607} C_VEL
LIN {X 0,Y 473.736,Z 359.354,A -85,B 0,C 180,E1 -7125.487,E2 -7125.487} C_VEL
LIN {X 0,Y 473.789,Z 358.267,A -85,B 0,C 180,E1 -7126.369,E2 -7126.369} C_VEL
LIN {X 0,Y 473.885,Z 355.451,A -85,B 0,C 180,E1 -7127.698,E2 -7127.698} C_VEL
LIN {X 0,Y 473.999,Z 352.621,A -85,B 0,C 180,E1 -7128.656,E2 -7128.656} C_VEL
LIN {X 0,Y 474.119,Z 349.59,A -85,B 0,C 180,E1 -7129.481,E2 -7129.481} C_VEL
LIN {X 0,Y 474.279,Z 344.315,A -85,B 0,C 180,E1 -7130.604,E2 -7130.604} C_VEL
LIN {X 0,Y 474.474,Z 339.059,A -85,B 0,C 180,E1 -7131.51,E2 -7131.51} C_VEL
LIN {X 0,Y 474.711,Z 332.708,A -85,B 0,C 180,E1 -7132.408,E2 -7132.408} C_VEL
LIN {X 0,Y 474.933,Z 325.7,A -85,B 0,C 180,E1 -7133.225,E2 -7133.225} C_VEL
LIN {X 0,Y 475.226,Z 317.601,A -85,B 0,C 180,E1 -7133.996,E2 -7133.996} C_VEL
LIN {X 0,Y 475.576,Z 308.712,A -85,B 0,C 180,E1 -7134.674,E2 -7134.674} C_VEL
LIN {X 0,Y 475.845,Z 298.381,A -85,B 0,C 180,E1 -7135.283,E2 -7135.283} C_VEL
LIN {X 0,Y 475.682,Z 292.316,A -85,B 0,C 180,E1 -7135.561,E2 -7135.561} C_VEL
LIN {X 0,Y 473.83,Z 282.103,A -85,B 0,C 180,E1 -7135.979,E2 -7135.979} C_VEL
LIN {X 0,Y 473.841,Z 277.663,A -85,B 0,C 180,E1 -7139.303,E2 -7139.303} C_VEL
LIN {X 0,Y 473.943,Z 273.695,A -85,B 0,C 180,E1 -7142.307,E2 -7142.307} C_VEL
LIN {X 0,Y 473.981,Z 269.767,A -85,B 0,C 180,E1 -7145.366,E2 -7145.366} C_VEL
LIN {X 0,Y 474.051,Z 265.755,A -85,B 0,C 180,E1 -7148.509,E2 -7148.509} C_VEL
LIN {X 0,Y 474.157,Z 261.61,A -85,B 0,C 180,E1 -7151.834,E2 -7151.834} C_VEL
LIN {X 0,Y 474.31,Z 258.219,A -85,B 0,C 180,E1 -7154.668,E2 -7154.668} C_VEL
LIN {X 0,Y 474.574,Z 258.184,A -85,B 0,C 180,E1 -7157.768,E2 -7157.768} C_VEL
LIN {X 0,Y 474.653,Z 258.172,A -85,B 0,C 180,E1 -7160.458,E2 -7160.458} C_VEL
LIN {X 0,Y 474.575,Z 258.183,A -85,B 0,C 180,E1 -7163.678,E2 -7163.678} C_VEL
LIN {X 0,Y 474.623,Z 258.176,A -85,B 0,C 180,E1 -7166.781,E2 -7166.781} C_VEL
LIN {X 0,Y 474.586,Z 258.18,A -85,B 0,C 180,E1 -7169.771,E2 -7169.771} C_VEL
LIN {X 0,Y 474.679,Z 258.169,A -85,B 0,C 180,E1 -7172.681,E2 -7172.681} C_VEL
LIN {X 0,Y 474.637,Z 258.176,A -85,B 0,C 180,E1 -7175.508,E2 -7175.508} C_VEL
LIN {X 0,Y 474.654,Z 258.17,A -85,B 0,C 180,E1 -7179.187,E2 -7179.187} C_VEL
LIN {X 0,Y 474.641,Z 258.174,A -85,B 0,C 180,E1 -7181.886,E2 -7181.886} C_VEL
LIN {X 0,Y 474.684,Z 258.17,A -85,B 0,C 180,E1 -7184.546,E2 -7184.546} C_VEL
LIN {X 0,Y 474.725,Z 258.167,A -85,B 0,C 180,E1 -7188.04,E2 -7188.04} C_VEL
LIN {X 0,Y 474.714,Z 258.166,A -85,B 0,C 180,E1 -7191.488,E2 -7191.488} C_VEL
LIN {X 0,Y 474.735,Z 258.161,A -85,B 0,C 180,E1 -7194.906,E2 -7194.906} C_VEL
LIN {X 0,Y 474.885,Z 258.145,A -85,B 0,C 180,E1 -7197.457,E2 -7197.457} C_VEL
LIN {X 0,Y 474.898,Z 258.141,A -85,B 0,C 180,E1 -7200.002,E2 -7200.002} C_VEL
LIN {X 0,Y 474.881,Z 258.145,A -85,B 0,C 180,E1 -7202.546,E2 -7202.546} C_VEL
LIN {X 0,Y 474.77,Z 258.155,A -85,B 0,C 180,E1 -7205.949,E2 -7205.949} C_VEL
LIN {X 0,Y 474.716,Z 258.168,A -85,B 0,C 180,E1 -7208.515,E2 -7208.515} C_VEL
LIN {X 0,Y 474.729,Z 258.165,A -85,B 0,C 180,E1 -7211.963,E2 -7211.963} C_VEL
LIN {X 0,Y 474.671,Z 258.169,A -85,B 0,C 180,E1 -7215.769,E2 -7215.769} C_VEL
LIN {X 0,Y 474.653,Z 258.171,A -85,B 0,C 180,E1 -7219.012,E2 -7219.012} C_VEL
LIN {X 0,Y 474.582,Z 258.181,A -85,B 0,C 180,E1 -7221.73,E2 -7221.73} C_VEL
LIN {X 0,Y 474.645,Z 258.178,A -85,B 0,C 180,E1 -7224.495,E2 -7224.495} C_VEL
LIN {X 0,Y 474.629,Z 258.178,A -85,B 0,C 180,E1 -7227.325,E2 -7227.325} C_VEL
LIN {X 0,Y 474.597,Z 258.181,A -85,B 0,C 180,E1 -7230.232,E2 -7230.232} C_VEL
LIN {X 0,Y 474.637,Z 258.176,A -85,B 0,C 180,E1 -7233.222,E2 -7233.222} C_VEL
LIN {X 0,Y 474.578,Z 258.183,A -85,B 0,C 180,E1 -7236.326,E2 -7236.326} C_VEL
LIN {X 0,Y 474.645,Z 258.174,A -85,B 0,C 180,E1 -7239.652,E2 -7239.652} C_VEL
LIN {X 0,Y 474.609,Z 258.179,A -85,B 0,C 180,E1 -7242.936,E2 -7242.936} C_VEL
LIN {X 0,Y 474.602,Z 258.179,A -85,B 0,C 180,E1 -7245.896,E2 -7245.896} C_VEL
LIN {X 0,Y 474.624,Z 258.177,A -85,B 0,C 180,E1 -7249.042,E2 -7249.042} C_VEL
LIN {X 0,Y 474.606,Z 258.183,A -85,B 0,C 180,E1 -7251.706,E2 -7251.706} C_VEL
LIN {X 0,Y 474.623,Z 258.374,A -85,B 0,C 180,E1 -7253.538,E2 -7253.538} C_VEL
LIN {X 0,Y 475.729,Z 264.486,A -85,B 0,C 180,E1 -7256.371,E2 -7256.371} C_VEL
LIN {X 0,Y 475.755,Z 269.124,A -85,B 0,C 180,E1 -7258.373,E2 -7258.373} C_VEL
LIN {X 0,Y 475.257,Z 277.531,A -85,B 0,C 180,E1 -7261.759,E2 -7261.759} C_VEL
LIN {X 0,Y 474.815,Z 286.057,A -85,B 0,C 180,E1 -7265.05,E2 -7265.05} C_VEL
LIN {X 0,Y 474.538,Z 293.442,A -85,B 0,C 180,E1 -7267.813,E2 -7267.813} C_VEL
LIN {X 0,Y 474.264,Z 302.138,A -85,B 0,C 180,E1 -7270.974,E2 -7270.974} C_VEL
LIN {X 0,Y 474.059,Z 312.134,A -85,B 0,C 180,E1 -7274.524,E2 -7274.524} C_VEL
LIN {X 0,Y 473.964,Z 322.272,A -85,B 0,C 180,E1 -7278.02,E2 -7278.02} C_VEL
LIN {X 0,Y 475.166,Z 334.356,A -85,B 0,C 180,E1 -7278.428,E2 -7278.428} C_VEL
LIN {X 0,Y 475.548,Z 341.298,A -85,B 0,C 180,E1 -7278.747,E2 -7278.747} C_VEL
LIN {X 0,Y 475.256,Z 351.701,A -85,B 0,C 180,E1 -7279.349,E2 -7279.349} C_VEL
LIN {X 0,Y 474.918,Z 360.253,A -85,B 0,C 180,E1 -7279.988,E2 -7279.988} C_VEL
LIN {X 0,Y 474.596,Z 368.314,A -85,B 0,C 180,E1 -7280.734,E2 -7280.734} C_VEL
LIN {X 0,Y 474.391,Z 374.984,A -85,B 0,C 180,E1 -7281.482,E2 -7281.482} C_VEL
LIN {X 0,Y 474.171,Z 381.323,A -85,B 0,C 180,E1 -7282.335,E2 -7282.335} C_VEL
LIN {X 0,Y 474.03,Z 386.596,A -85,B 0,C 180,E1 -7283.189,E2 -7283.189} C_VEL
LIN {X 0,Y 473.925,Z 390.998,A -85,B 0,C 180,E1 -7284.043,E2 -7284.043} C_VEL
LIN {X 0,Y 473.791,Z 396.197,A -85,B 0,C 180,E1 -7285.322,E2 -7285.322} C_VEL
LIN {X 0,Y 473.845,Z 400.023,A -85,B 0,C 180,E1 -7286.6,E2 -7286.6} C_VEL
LIN {X 0,Y 473.765,Z 401.778,A -85,B 0,C 180,E1 -7287.45,E2 -7287.45} C_VEL
LIN {X 0,Y 473.756,Z 403.036,A -85,B 0,C 180,E1 -7288.301,E2 -7288.301} C_VEL
LIN {X 0,Y 473.689,Z 403.817,A -85,B 0,C 180,E1 -7289.151,E2 -7289.151} C_VEL
LIN {X 0,Y 473.674,Z 404.115,A -85,B 0,C 180,E1 -7290.001,E2 -7290.001} C_VEL
LIN {X 0,Y 473.689,Z 403.819,A -85,B 0,C 180,E1 -7290.851,E2 -7290.851} C_VEL
LIN {X 0,Y 473.756,Z 403.034,A -85,B 0,C 180,E1 -7291.701,E2 -7291.701} C_VEL
LIN {X 0,Y 473.766,Z 401.768,A -85,B 0,C 180,E1 -7292.552,E2 -7292.552} C_VEL
LIN {X 0,Y 473.828,Z 398.846,A -85,B 0,C 180,E1 -7293.828,E2 -7293.828} C_VEL
LIN {X 0,Y 473.792,Z 396.173,A -85,B 0,C 180,E1 -7294.681,E2 -7294.681} C_VEL
LIN {X 0,Y 473.927,Z 390.959,A -85,B 0,C 180,E1 -7295.959,E2 -7295.959} C_VEL
LIN {X 0,Y 474.126,Z 384.076,A -85,B 0,C 180,E1 -7297.239,E2 -7297.239} C_VEL
LIN {X 0,Y 474.324,Z 376.556,A -85,B 0,C 180,E1 -7298.307,E2 -7298.307} C_VEL
LIN {X 0,Y 474.558,Z 369.136,A -85,B 0,C 180,E1 -7299.162,E2 -7299.162} C_VEL
LIN {X 0,Y 474.841,Z 361.189,A -85,B 0,C 180,E1 -7299.909,E2 -7299.909} C_VEL
LIN {X 0,Y 475.239,Z 351.283,A -85,B 0,C 180,E1 -7300.654,E2 -7300.654} C_VEL
LIN {X 0,Y 475.514,Z 340.604,A -85,B 0,C 180,E1 -7301.251,E2 -7301.251} C_VEL
LIN {X 0,Y 474.765,Z 330.498,A -85,B 0,C 180,E1 -7301.678,E2 -7301.678} C_VEL
LIN {X 0,Y 473.926,Z 322.27,A -85,B 0,C 180,E1 -7301.948,E2 -7301.948} C_VEL
LIN {X 0,Y 474.06,Z 312.018,A -85,B 0,C 180,E1 -7305.498,E2 -7305.498} C_VEL
LIN {X 0,Y 474.231,Z 303.551,A -85,B 0,C 180,E1 -7308.473,E2 -7308.473} C_VEL
LIN {X 0,Y 474.473,Z 294.397,A -85,B 0,C 180,E1 -7311.735,E2 -7311.735} C_VEL
LIN {X 0,Y 474.791,Z 285.572,A -85,B 0,C 180,E1 -7314.953,E2 -7314.953} C_VEL
LIN {X 0,Y 475.144,Z 276.767,A -85,B 0,C 180,E1 -7318.251,E2 -7318.251} C_VEL
LIN {X 0,Y 475.54,Z 269.249,A -85,B 0,C 180,E1 -7321.15,E2 -7321.15} C_VEL
LIN {X 0,Y 475.639,Z 264.26,A -85,B 0,C 180,E1 -7323.142,E2 -7323.142} C_VEL
LIN {X 0,Y 474.637,Z 258.178,A -85,B 0,C 180,E1 -7325.752,E2 -7325.752} C_VEL
LIN {X 0,Y 474.619,Z 258.18,A -85,B 0,C 180,E1 -7328.458,E2 -7328.458} C_VEL
LIN {X 0,Y 474.628,Z 258.178,A -85,B 0,C 180,E1 -7331.786,E2 -7331.786} C_VEL
LIN {X 0,Y 474.625,Z 258.177,A -85,B 0,C 180,E1 -7335.298,E2 -7335.298} C_VEL
LIN {X 0,Y 474.629,Z 258.179,A -85,B 0,C 180,E1 -7338.214,E2 -7338.214} C_VEL
LIN {X 0,Y 474.618,Z 258.18,A -85,B 0,C 180,E1 -7341.542,E2 -7341.542} C_VEL
LIN {X 0,Y 474.63,Z 258.177,A -85,B 0,C 180,E1 -7344.725,E2 -7344.725} C_VEL
LIN {X 0,Y 474.644,Z 258.176,A -85,B 0,C 180,E1 -7347.787,E2 -7347.787} C_VEL
LIN {X 0,Y 474.632,Z 258.178,A -85,B 0,C 180,E1 -7350.884,E2 -7350.884} C_VEL
LIN {X 0,Y 474.663,Z 258.175,A -85,B 0,C 180,E1 -7353.627,E2 -7353.627} C_VEL
LIN {X 0,Y 474.644,Z 258.175,A -85,B 0,C 180,E1 -7356.641,E2 -7356.641} C_VEL
LIN {X 0,Y 474.663,Z 258.171,A -85,B 0,C 180,E1 -7360.089,E2 -7360.089} C_VEL
LIN {X 0,Y 474.646,Z 258.176,A -85,B 0,C 180,E1 -7362.773,E2 -7362.773} C_VEL
LIN {X 0,Y 474.655,Z 258.175,A -85,B 0,C 180,E1 -7365.42,E2 -7365.42} C_VEL
LIN {X 0,Y 474.712,Z 258.166,A -85,B 0,C 180,E1 -7368.036,E2 -7368.036} C_VEL
LIN {X 0,Y 474.718,Z 258.167,A -85,B 0,C 180,E1 -7371.485,E2 -7371.485} C_VEL
LIN {X 0,Y 474.776,Z 258.159,A -85,B 0,C 180,E1 -7374.051,E2 -7374.051} C_VEL
LIN {X 0,Y 474.899,Z 258.143,A -85,B 0,C 180,E1 -7377.454,E2 -7377.454} C_VEL
LIN {X 0,Y 474.917,Z 258.142,A -85,B 0,C 180,E1 -7379.998,E2 -7379.998} C_VEL
LIN {X 0,Y 474.899,Z 258.144,A -85,B 0,C 180,E1 -7382.543,E2 -7382.543} C_VEL
LIN {X 0,Y 474.783,Z 258.158,A -85,B 0,C 180,E1 -7385.946,E2 -7385.946} C_VEL
LIN {X 0,Y 474.732,Z 258.165,A -85,B 0,C 180,E1 -7388.512,E2 -7388.512} C_VEL
LIN {X 0,Y 474.707,Z 258.168,A -85,B 0,C 180,E1 -7391.961,E2 -7391.961} C_VEL
LIN {X 0,Y 474.702,Z 258.168,A -85,B 0,C 180,E1 -7395.454,E2 -7395.454} C_VEL
LIN {X 0,Y 474.666,Z 258.172,A -85,B 0,C 180,E1 -7399.008,E2 -7399.008} C_VEL
LIN {X 0,Y 474.589,Z 258.183,A -85,B 0,C 180,E1 -7401.727,E2 -7401.727} C_VEL
LIN {X 0,Y 474.658,Z 258.173,A -85,B 0,C 180,E1 -7404.491,E2 -7404.491} C_VEL
LIN {X 0,Y 474.697,Z 258.17,A -85,B 0,C 180,E1 -7407.336,E2 -7407.336} C_VEL
LIN {X 0,Y 474.602,Z 258.179,A -85,B 0,C 180,E1 -7410.808,E2 -7410.808} C_VEL
LIN {X 0,Y 474.634,Z 258.178,A -85,B 0,C 180,E1 -7413.982,E2 -7413.982} C_VEL
LIN {X 0,Y 474.569,Z 258.184,A -85,B 0,C 180,E1 -7416.898,E2 -7416.898} C_VEL
LIN {X 0,Y 474.643,Z 258.176,A -85,B 0,C 180,E1 -7419.649,E2 -7419.649} C_VEL
LIN {X 0,Y 474.644,Z 258.176,A -85,B 0,C 180,E1 -7422.928,E2 -7422.928} C_VEL
LIN {X 0,Y 474.609,Z 258.179,A -85,B 0,C 180,E1 -7425.894,E2 -7425.894} C_VEL
LIN {X 0,Y 474.637,Z 258.177,A -85,B 0,C 180,E1 -7429.036,E2 -7429.036} C_VEL
LIN {X 0,Y 474.609,Z 258.179,A -85,B 0,C 180,E1 -7431.7,E2 -7431.7} C_VEL
LIN {X 0,Y 474.619,Z 258.18,A -85,B 0,C 180,E1 -7434.724,E2 -7434.724} C_VEL
LIN {X 0,Y 474.625,Z 258.177,A -85,B 0,C 180,E1 -7437.786,E2 -7437.786} C_VEL
LIN {X 0,Y 474.618,Z 258.18,A -85,B 0,C 180,E1 -7440.881,E2 -7440.881} C_VEL
LIN {X 0,Y 474.652,Z 258.174,A -85,B 0,C 180,E1 -7443.627,E2 -7443.627} C_VEL
LIN {X 0,Y 474.626,Z 258.18,A -85,B 0,C 180,E1 -7446.638,E2 -7446.638} C_VEL
LIN {X 0,Y 474.659,Z 258.173,A -85,B 0,C 180,E1 -7449.184,E2 -7449.184} C_VEL
LIN {X 0,Y 474.566,Z 258.184,A -85,B 0,C 180,E1 -7451.655,E2 -7451.655} C_VEL
LIN {X 0,Y 473.82,Z 258.284,A -85,B 0,C 180,E1 -7452.362,E2 -7452.362} C_VEL
LIN {X 0,Y 470.832,Z 258.665,A -85,B 0,C 180,E1 -7453.507,E2 -7453.507} C_VEL
LIN {X 0,Y 468.326,Z 259.324,A -85,B 0,C 180,E1 -7454.427,E2 -7454.427} C_VEL
LIN {X 0,Y 467.234,Z 260.054,A -85,B 0,C 180,E1 -7455.136,E2 -7455.136} C_VEL
LIN {X 0,Y 467.136,Z 260.347,A -85,B 0,C 180,E1 -7455.376,E2 -7455.376} C_VEL
LIN {X 0,Y 467.2,Z 263.557,A -85,B 0,C 180,E1 -7457.887,E2 -7457.887} C_VEL
LIN {X 0,Y 467.038,Z 268.043,A -85,B 0,C 180,E1 -7461.344,E2 -7461.344} C_VEL
LIN {X 0,Y 467.035,Z 271.437,A -85,B 0,C 180,E1 -7463.952,E2 -7463.952} C_VEL
LIN {X 0,Y 467.03,Z 274.872,A -85,B 0,C 180,E1 -7466.548,E2 -7466.548} C_VEL
LIN {X 0,Y 466.712,Z 279.529,A -85,B 0,C 180,E1 -7469.999,E2 -7469.999} C_VEL
LIN {X 0,Y 466.726,Z 282.229,A -85,B 0,C 180,E1 -7471.994,E2 -7471.994} C_VEL
LIN {X 0,Y 468.732,Z 293.496,A -85,B 0,C 180,E1 -7472.469,E2 -7472.469} C_VEL
LIN {X 0,Y 468.62,Z 302.147,A -85,B 0,C 180,E1 -7472.9,E2 -7472.9} C_VEL
LIN {X 0,Y 468.367,Z 310.627,A -85,B 0,C 180,E1 -7473.44,E2 -7473.44} C_VEL
LIN {X 0,Y 468.062,Z 318.787,A -85,B 0,C 180,E1 -7474.089,E2 -7474.089} C_VEL
LIN {X 0,Y 467.79,Z 326.524,A -85,B 0,C 180,E1 -7474.847,E2 -7474.847} C_VEL
LIN {X 0,Y 467.612,Z 332.904,A -85,B 0,C 180,E1 -7475.605,E2 -7475.605} C_VEL
LIN {X 0,Y 467.404,Z 339.909,A -85,B 0,C 180,E1 -7476.614,E2 -7476.614} C_VEL
LIN {X 0,Y 467.166,Z 346.353,A -85,B 0,C 180,E1 -7477.78,E2 -7477.78} C_VEL
LIN {X 0,Y 466.967,Z 350.209,A -85,B 0,C 180,E1 -7478.655,E2 -7478.655} C_VEL
LIN {X 0,Y 466.833,Z 354.645,A -85,B 0,C 180,E1 -7479.969,E2 -7479.969} C_VEL
LIN {X 0,Y 466.706,Z 358.738,A -85,B 0,C 180,E1 -7481.827,E2 -7481.827} C_VEL
LIN {X 0,Y 466.615,Z 360.077,A -85,B 0,C 180,E1 -7483.056,E2 -7483.056} C_VEL
LIN {X 0,Y 466.594,Z 360.414,A -85,B 0,C 180,E1 -7483.944,E2 -7483.944} C_VEL
LIN {X 0,Y 466.659,Z 359.75,A -85,B 0,C 180,E1 -7485.462,E2 -7485.462} C_VEL
LIN {X 0,Y 466.724,Z 358.215,A -85,B 0,C 180,E1 -7486.624,E2 -7486.624} C_VEL
LIN {X 0,Y 466.846,Z 355.236,A -85,B 0,C 180,E1 -7487.974,E2 -7487.974} C_VEL
LIN {X 0,Y 466.949,Z 352.469,A -85,B 0,C 180,E1 -7488.879,E2 -7488.879} C_VEL
LIN {X 0,Y 467.092,Z 349.005,A -85,B 0,C 180,E1 -7489.787,E2 -7489.787} C_VEL
LIN {X 0,Y 467.227,Z 344.743,A -85,B 0,C 180,E1 -7490.699,E2 -7490.699} C_VEL
LIN {X 0,Y 467.429,Z 339.839,A -85,B 0,C 180,E1 -7491.567,E2 -7491.567} C_VEL
LIN {X 0,Y 467.696,Z 333.182,A -85,B 0,C 180,E1 -7492.53,E2 -7492.53} C_VEL
LIN {X 0,Y 467.953,Z 326.187,A -85,B 0,C 180,E1 -7493.36,E2 -7493.36} C_VEL
LIN {X 0,Y 468.221,Z 319.453,A -85,B 0,C 180,E1 -7494.024,E2 -7494.024} C_VEL
LIN {X 0,Y 468.516,Z 312.494,A -85,B 0,C 180,E1 -7494.598,E2 -7494.598} C_VEL
LIN {X 0,Y 468.783,Z 304.352,A -85,B 0,C 180,E1 -7495.145,E2 -7495.145} C_VEL
LIN {X 0,Y 468.98,Z 295.646,A -85,B 0,C 180,E1 -7495.606,E2 -7495.606} C_VEL
LIN {X 0,Y 467.658,Z 287.105,A -85,B 0,C 180,E1 -7495.993,E2 -7495.993} C_VEL
LIN {X 0,Y 466.76,Z 282.396,A -85,B 0,C 180,E1 -7496.201,E2 -7496.201} C_VEL
LIN {X 0,Y 466.789,Z 277.654,A -85,B 0,C 180,E1 -7499.79,E2 -7499.79} C_VEL
LIN {X 0,Y 466.864,Z 273.716,A -85,B 0,C 180,E1 -7502.813,E2 -7502.813} C_VEL
LIN {X 0,Y 466.933,Z 269.728,A -85,B 0,C 180,E1 -7505.943,E2 -7505.943} C_VEL
LIN {X 0,Y 467.016,Z 265.675,A -85,B 0,C 180,E1 -7509.199,E2 -7509.199} C_VEL
LIN {X 0,Y 467.167,Z 261.467,A -85,B 0,C 180,E1 -7512.606,E2 -7512.606} C_VEL
LIN {X 0,Y 467.22,Z 260.04,A -85,B 0,C 180,E1 -7513.782,E2 -7513.782} C_VEL
LIN {X 0,Y 467.296,Z 259.091,A -85,B 0,C 180,E1 -7515.023,E2 -7515.023} C_VEL
LIN {X 0,Y 467.501,Z 259.062,A -85,B 0,C 180,E1 -7517.442,E2 -7517.442} C_VEL
LIN {X 0,Y 467.582,Z 259.053,A -85,B 0,C 180,E1 -7520.043,E2 -7520.043} C_VEL
LIN {X 0,Y 467.515,Z 259.064,A -85,B 0,C 180,E1 -7523.039,E2 -7523.039} C_VEL
LIN {X 0,Y 467.567,Z 259.056,A -85,B 0,C 180,E1 -7526.213,E2 -7526.213} C_VEL
LIN {X 0,Y 467.55,Z 259.059,A -85,B 0,C 180,E1 -7529.267,E2 -7529.267} C_VEL
LIN {X 0,Y 467.626,Z 259.049,A -85,B 0,C 180,E1 -7532.46,E2 -7532.46} C_VEL
LIN {X 0,Y 467.577,Z 259.056,A -85,B 0,C 180,E1 -7535.113,E2 -7535.113} C_VEL
LIN {X 0,Y 467.517,Z 259.061,A -85,B 0,C 180,E1 -7537.927,E2 -7537.927} C_VEL
LIN {X 0,Y 467.608,Z 259.049,A -85,B 0,C 180,E1 -7540.694,E2 -7540.694} C_VEL
LIN {X 0,Y 467.634,Z 259.046,A -85,B 0,C 180,E1 -7544.116,E2 -7544.116} C_VEL
LIN {X 0,Y 467.669,Z 259.045,A -85,B 0,C 180,E1 -7547.857,E2 -7547.857} C_VEL
LIN {X 0,Y 467.668,Z 259.045,A -85,B 0,C 180,E1 -7551.359,E2 -7551.359} C_VEL
LIN {X 0,Y 467.706,Z 259.037,A -85,B 0,C 180,E1 -7554.829,E2 -7554.829} C_VEL
LIN {X 0,Y 467.85,Z 259.021,A -85,B 0,C 180,E1 -7557.419,E2 -7557.419} C_VEL
LIN {X 0,Y 467.869,Z 259.017,A -85,B 0,C 180,E1 -7560.002,E2 -7560.002} C_VEL
